// TIA Portal project "KumKoprusu" (V15)

(* hardware
DEVICE "S7-1200 station_1"  S7-1200 Station
   slot 0: "Rack_0"  S7-1200 Rack  Rack  V1.0
   slot 1: "KumKoprusu"  CPU 1214C DC/DC/Rly  6ES7 214-1HG40-0XB0  V4.2
   slot 2: "DI 16x24VDC/DQ 16xRelay_1"  SM 1223 DI16/DQ16 x relay  6ES7 223-1PL32-0XB0  V2.0
*)

// ===== PLC "KumKoprusu"  CPU 1214C DC/DC/Rly =====

VAR_GLOBAL   // PLC tag table "Default tag table"
   "SN_PULS" AT %M2.0 : Bool;
   "SN" AT %MW4 : Int;
   "DK_PULSE" AT %M2.1 : Bool;
END_VAR

VAR_GLOBAL   // PLC tag table "Input"
   "KPR_ACLSTP" AT %I0.0 : Bool;
   "KPR_ILERI_MAN/OTO" AT %I0.1 : Bool;
   "KPR_GERI_MAN/OTO" AT %I0.4 : Bool;
   "KPR_BASTA" AT %I0.7 : Bool;
   "KPR_SONDA" AT %I1.0 : Bool;
   "SYR1_MAN/OTO" AT %I1.1 : Bool;
   "SYR1_YKRD" AT %I1.4 : Bool;
   "SYR1_ASGD" AT %I1.5 : Bool;
   "SYR2_MAN/OTO" AT %I2.0 : Bool;
   "SYR2_YKRD" AT %I2.3 : Bool;
   "SYR2_ASGD" AT %I2.4 : Bool;
   "KPR_GERI_ARZ" AT %I0.6 : Bool;
   "P1_MAN/OTO" AT %I2.5 : Bool;
   "P1_DVRD" AT %I2.6 : Bool;
   "P1_ARZ" AT %I2.7 : Bool;
   "P2_MAN/OTO" AT %I3.0 : Bool;
   "P2_DVRD" AT %I3.1 : Bool;
   "P2_ARZ" AT %I3.2 : Bool;
   "SYR1_DVRD" AT %I1.2 : Bool;
   "SYR1_ARZ" AT %I1.3 : Bool;
   "SYR2_DVRD" AT %I2.1 : Bool;
   "SYR2_ARZ" AT %I2.2 : Bool;
   "KPR_ILERI_ARZ" AT %I0.3 : Bool;
   "KPR_ILERI_DVRD" AT %I0.2 : Bool;
   "KPR_GERI_DVRD" AT %I0.5 : Bool;
END_VAR

VAR_GLOBAL   // PLC tag table "Output"
   "KPR_ILERI_RUNQ" AT %Q0.0 : Bool;
   "KPR_GERI_RUNQ" AT %Q0.1 : Bool;
   "SYR1_ASG_RUNQ" AT %Q0.2 : Bool;
   "SYR1_YKR_RUNQ" AT %Q0.3 : Bool;
   "SYR2_ASG_RUNQ" AT %Q0.4 : Bool;
   "SYR2_YKR_RUNQ" AT %Q0.5 : Bool;
   "P1_RUNQ" AT %Q1.0 : Bool;
   "P2_RUNQ" AT %Q1.1 : Bool;
END_VAR

VAR_GLOBAL   // PLC tag table "Flag"
   "System_Byte" AT %MB1 : Byte;
   "FirstScan" AT %M1.0 : Bool;
   "DiagStatusUpdate" AT %M1.1 : Bool;
   "AlwaysTRUE" AT %M1.2 : Bool;
   "AlwaysFALSE" AT %M1.3 : Bool;
   "Clock_Byte" AT %MB0 : Byte;
   "Clock_10Hz" AT %M0.0 : Bool;
   "Clock_5Hz" AT %M0.1 : Bool;
   "Clock_2.5Hz" AT %M0.2 : Bool;
   "Clock_2Hz" AT %M0.3 : Bool;
   "Clock_1.25Hz" AT %M0.4 : Bool;
   "Clock_1Hz" AT %M0.5 : Bool;
   "Clock_0.625Hz" AT %M0.6 : Bool;
   "Clock_0.5Hz" AT %M0.7 : Bool;
END_VAR

// folder: DB

DATA_BLOCK "KOPRU_DB"   // DB1
{ S7_Optimized_Access := 'TRUE' }
VERSION : 0.1
// stored: InstanceOfName KOPRU_FB
"KOPRU_FB"
BEGIN
END_DATA_BLOCK

DATA_BLOCK "FB_I/O"   // DB2
{ S7_Optimized_Access := 'FALSE' }
VERSION : 0.1
   VAR
      KPR_SCD_RESET : Bool;
      "KPR_SCD_MAN/OTO" : Bool;
      KPR_SCD_MAN_İLERİ : Bool;
      KPR_SCD_MAN_GERİ : Bool;
      SYR_SCD_RESET : Bool;
      "SYR1_SCD_MAN/OTO" : Bool;
      SYR1_SCD_MAN_ASAGI : Bool;
      SYR1_SCD_MAN_YUKARI : Bool;
      "SYR2_SCD_MAN/OTO" : Bool;
      SYR2_SCD_MAN_ASAGI : Bool;
      SYR2_SCD_MAN_YUKARI : Bool;
      "P1_SCD_MAN/OTO" : Bool;
      P1_SCD_MAN_CALIS : Bool;
      "P2_SCD_MAN/OTO" : Bool;
      P2_SCD_MAN_CALIS : Bool;
      Q_KPR_ACIL_STOP : Bool;
      Q_KPR_OTO : Bool;
      Q_KPR_ILERI_GDYR : Bool;
      Q_KPR_SONDA : Bool;
      Q_KPR_GERI_GDYR : Bool;
      Q_KPR_BASTA : Bool;
      Q_KPR_ARIZA : Bool;
      Q_KPR_GECIKME_HATA : Bool;
      Q_KPR_SWITCH_HATA : Bool;
      Q_SYR1_OTO : Bool;
      Q_SYR1_DVRD : Bool;
      Q_SYR1_ASAGIDA : Bool;
      Q_SYR1_YUKARIDA : Bool;
      Q_SYR1_ARIZA : Bool;
      Q_SYR1_GECIKME_HATA : Bool;
      Q_SYR1_SWITCH_HATA : Bool;
      Q_SYR2_OTO : Bool;
      Q_SYR2_DVRD : Bool;
      Q_SYR2_ASAGIDA : Bool;
      Q_SYR2_YUKARIDA : Bool;
      Q_SYR2_ARIZA : Bool;
      Q_SYR2_GECIKME_HATA : Bool;
      Q_SYR2_SWITCH_HATA : Bool;
      Q_P1_OTO : Bool;
      Q_P1_CALISIYOR : Bool;
      Q_P1_ARIZA : Bool;
      Q_P2_OTO : Bool;
      Q_P2_CALISIYOR : Bool;
      Q_P2_ARIZA : Bool;
      Q_PARK_KALAN_SURE : Int;
      Q_IST_KALAN_SURE : Int;
      Q_KPR_SAAT : DInt;
      Q_KPR_DK : DInt;
      Q_KPR_BAKIM_ZAM_FARK : DInt;
      Q_SYR1_SAAT : DInt;
      Q_SYR1_DK : DInt;
      Q_SYR1_BAKIM_ZAM_FARK : DInt;
      Q_SYR2_SAAT : DInt;
      Q_SYR2_DK : DInt;
      Q_SYR2_BAKIM_ZAM_FARK : DInt;
   END_VAR
BEGIN
END_DATA_BLOCK

// folder: (top level)

ORGANIZATION_BLOCK "Main"   // OB1, LAD, ProgramCycle
TITLE = "Main Program Sweep (Cycle)"
{ S7_Optimized_Access := 'TRUE' }
VERSION : 0.1
   VAR_INPUT
      Initial_Call : Bool;   // Initial call of this OB
      Remanence : Bool;   // =True, if remanent data are available
   END_VAR
   VAR_TEMP   // added for the SCL form of the ladder/FBD networks
      _w1 : Bool;
      _w2 : Bool;
   END_VAR
BEGIN

REGION Network 1
   // SN PULSE
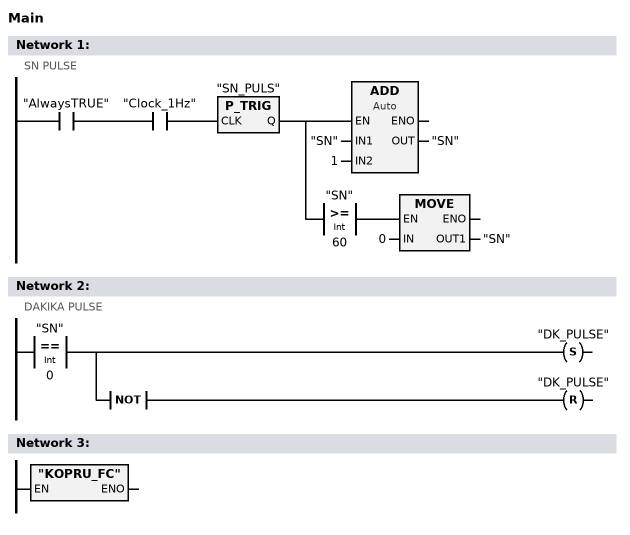
   RUNG wire#powerrail
      Contact( "AlwaysTRUE" )
      Contact( "Clock_1Hz" )
      P_Trig( "SN_PULS" )
      wire#w1
      Add(in1 := "SN", in2 := 1, out => "SN")
   END_RUNG
   RUNG wire#w1
      { S7_Templates := "SrcType := Int" } GE_Contact(in1 := "SN", in2 := 60)
      Move(in := 0, out1 => "SN")
   END_RUNG
   // the same network as SCL:
   #_w1 := "AlwaysTRUE" AND "Clock_1Hz";
   #_w2 := #_w1 AND NOT "SN_PULS";   // rising edge
   "SN_PULS" := #_w1;
   IF #_w2 THEN "SN" := "SN" + 1; END_IF;
   IF #_w2 AND ("SN" >= 60) THEN "SN" := 0; END_IF;
END_REGION

REGION Network 2
   // DAKIKA PULSE
   RUNG wire#powerrail
      { S7_Templates := "SrcType := Int" } EQ_Contact(in1 := "SN", in2 := 0)
      wire#w1
      S_Coil( "DK_PULSE" )
   END_RUNG
   RUNG wire#w1
      Not()
      R_Coil( "DK_PULSE" )
   END_RUNG
   // the same network as SCL:
   #_w1 := "SN" = 0;
   IF #_w1 THEN "DK_PULSE" := TRUE; END_IF;
   IF NOT #_w1 THEN "DK_PULSE" := FALSE; END_IF;
END_REGION

REGION Network 3
   RUNG wire#powerrail
      "KOPRU_FC"()
   END_RUNG
   // the same network as SCL:
   "KOPRU_FC"();
END_REGION
END_ORGANIZATION_BLOCK

// folder: FB

FUNCTION_BLOCK "KOPRU_FB"   // FB1, LAD
{ S7_Optimized_Access := 'TRUE' }
VERSION : 0.1
   VAR_INPUT
      KPR_ACLSTP : Bool;
      KPR_RESET : Bool;
      "KPR_SCADA_MAN/OTO" : Bool;
      "KPR_ILERI_MAN/OTO" : Bool;
      KPR_ILERI_DVRD : Bool;
      KPR_ILERI_ARZ : Bool;
      "KPR_GERI_MAN/OTO" : Bool;
      KPR_GERI_DVRD : Bool;
      KPR_GERI_ARZ : Bool;
      KPR_BASTA : Bool;
      KPR_SONDA : Bool;
      KPR_MAN_İLERİ : Bool;
      KPR_MAN_GERİ : Bool;
      KPR_BAKIM_ZAM_SET : DInt;
      SYR_RESET : Bool;
      "SYR1_SCADA_MAN/OTO" : Bool;
      "SYR1_MAN/OTO" : Bool;
      SYR1_DVRD : Bool;
      SYR1_ARZ : Bool;
      SYR1_YKRD : Bool;
      SYR1_ASGD : Bool;
      SYR1_MAN_ASAGI : Bool;
      SYR1_MAN_YUKARI : Bool;
      "SYR2_SCADA_MAN/OTO" : Bool;
      "SYR2_MAN/OTO" : Bool;
      SYR2_DVRD : Bool;
      SYR2_ARZ : Bool;
      SYR2_YKRD : Bool;
      SYR2_ASGD : Bool;
      SYR2_MAN_ASAGI : Bool;
      SYR2_MAN_YUKARI : Bool;
      SYR_BAKIM_ZAM_SET : DInt;
      "P1_SCADA_MAN/OTO" : Bool;
      "P1_MAN/OTO" : Bool;
      P1_DVRD : Bool;
      P1_ARZ : Bool;
      P1_MAN_CALIS : Bool;
      "P2_SCADA_MAN/OTO" : Bool;
      "P2_MAN/OTO" : Bool;
      P2_DVRD : Bool;
      P2_ARZ : Bool;
      P2_MAN_CALIS : Bool;
      DAKIKA_PULSE : Bool;
      SANIYE_PULSE : Bool;
      "PARK_BEKLEME_SURESI(DK)" : Int;
      "ISTASYON_BEKLEME_SURESI(DK)" : Int;
      "GECIKME_HATASI(SN)" : Int;
   END_VAR
   VAR_OUTPUT
      Q_KPR_ACIL_STOP : Bool;
      Q_KPR_OTO : Bool;
      Q_KPR_ILERI_GIT : Bool;
      Q_KPR_GERI_GIT : Bool;
      Q_KPR_ILERI_GDYR : Bool;
      Q_KPR_SONDA : Bool;
      Q_KPR_GERI_GDYR : Bool;
      Q_KPR_BASTA : Bool;
      Q_KPR_ARIZA : Bool;
      Q_KPR_GECIKME_HATA : Bool;
      Q_KPR_SWITCH_HATA : Bool;
      Q_SYR1_OTO : Bool;
      Q_SYR1_ASAGI_GIT : Bool;
      Q_SYR1_YUKARI_GIT : Bool;
      Q_SYR1_DVRD : Bool;
      Q_SYR1_ASAGIDA : Bool;
      Q_SYR1_YUKARIDA : Bool;
      Q_SYR1_ARIZA : Bool;
      Q_SYR1_GECIKME_HATA : Bool;
      Q_SYR1_SWITCH_HATA : Bool;
      Q_SYR2_OTO : Bool;
      Q_SYR2_ASAGI_GIT : Bool;
      Q_SYR2_YUKARI_GIT : Bool;
      Q_SYR2_DVRD : Bool;
      Q_SYR2_ASAGIDA : Bool;
      Q_SYR2_YUKARIDA : Bool;
      Q_SYR2_ARIZA : Bool;
      Q_SYR2_GECIKME_HATA : Bool;
      Q_SYR2_SWITCH_HATA : Bool;
      Q_P1_OTO : Bool;
      Q_P1_CALIS : Bool;
      Q_P1_CALISIYOR : Bool;
      Q_P1_ARIZA : Bool;
      Q_P2_OTO : Bool;
      Q_P2_CALIS : Bool;
      Q_P2_CALISIYOR : Bool;
      Q_P2_ARIZA : Bool;
      Q_PARK_KALAN_SURE : Int;
      Q_IST_KALAN_SURE : Int;
      Q_KPR_SAAT : DInt;
      Q_KPR_DK : DInt;
      Q_KPR_BAKIM_ZAM_FARK : DInt;
      Q_SYR1_BAKIM_ZAM_FARK : DInt;
      Q_SYR1_SAAT : DInt;
      Q_SYR1_DK : DInt;
      Q_SYR2_BAKIM_ZAM_FARK : DInt;
      Q_SYR2_SAAT : DInt;
      Q_SYR2_DK : DInt;
   END_VAR
   VAR
      ALWAYS_ON : Bool;
      SISTEM_OTO_CLSBLR : Bool;
      SISTEM_OTO : Bool;
      "KPR_MAN/OTO" : Bool;
      KPR_ARIZA : Bool;
      KPR_GENEL_HATA : Bool;
      ILERI_GIT : Bool;
      GERI_GIT : Bool;
      ASAGI_GIT : Bool;
      YUKARI_GIT : Bool;
      "SYR_SCADA_MAN/OTO" : Bool;
      "SYR_MAN/OTO" : Bool;
      PARK_SURE_OK : Bool;
      PARK_SURE : Int;
      SYR1_ZAMAN : Int;
      KPR_ZAMAN : Int;
      SYR_GENEL_HATA : Bool;
      NEGATIF_KENAR_1 : Bool;
      NEGATIF_KENAR_2 : Bool;
      NEGATIF_KENAR_3 : Bool;
      NEGATIF_KENAR_4 : Bool;
      NEGATIF_KENAR_5 : Bool;
      POZ_1 : Bool;
      POZ_2 : Bool;
      POZ_3 : Bool;
      SAAT : DInt;
      DAKIKA : DInt;
      SANIYE : DInt;
      SAAT_1 : DInt;
      DAKIKA_1 : DInt;
      SANIYE_1 : DInt;
      SAAT_2 : DInt;
      DAKIKA_2 : DInt;
      SANIYE_2 : DInt;
      ISTASYON_SURE : Int;
      IST_SURE_OK : Bool;
      P2_CALIS : Bool;
      P1_CALIS : Bool;
   END_VAR
   VAR_TEMP
      KPR_CALISYOR : Bool;
      KPR_ILERI_CALIS : Bool;
      KPR_GERI_CALIS : Bool;
      SYR_CALISIYOR : Bool;
      SYR_ASAGIDA : Bool;
      SYR_YUKARDA : Bool;
      SYR1_ASAGI_CALIS : Bool;
      SYR1_YUKARI_CALIS : Bool;
      SYR2_ASAGI_CALIS : Bool;
      SYR2_YUKARI_CALIS : Bool;
      KPR_SWITCH_HATA : Bool;
      SYR1_SWITCH_HATA : Bool;
      SYR2_SWITCH_HATA : Bool;
      KPR_GECIKME_HATA : Bool;
      SYR1_GECIKME_HATA : Bool;
      SYR2_GECIKME_HATA : Bool;
      IPTAL_BITI : Bool;
      SYR2_ZAMAN : DInt;
   END_VAR
   VAR_TEMP   // added for the SCL form of the ladder/FBD networks
      _w1 : Bool;
      _w2 : Bool;
      _w3 : Bool;
   END_VAR
BEGIN

REGION Network 1
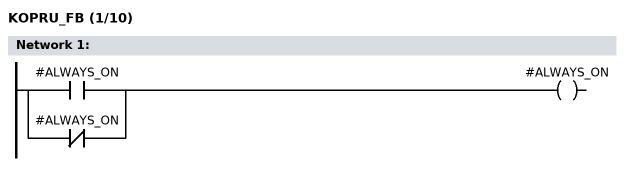
   RUNG wire#powerrail
      Contact( #ALWAYS_ON )
      wire#w1
      Coil( #ALWAYS_ON )
   END_RUNG
   RUNG wire#powerrail
      I_Contact( #ALWAYS_ON )
   END_RUNG wire#w1
   // the same network as SCL:
   #ALWAYS_ON := #ALWAYS_ON OR NOT #ALWAYS_ON;
END_REGION

REGION Network 2
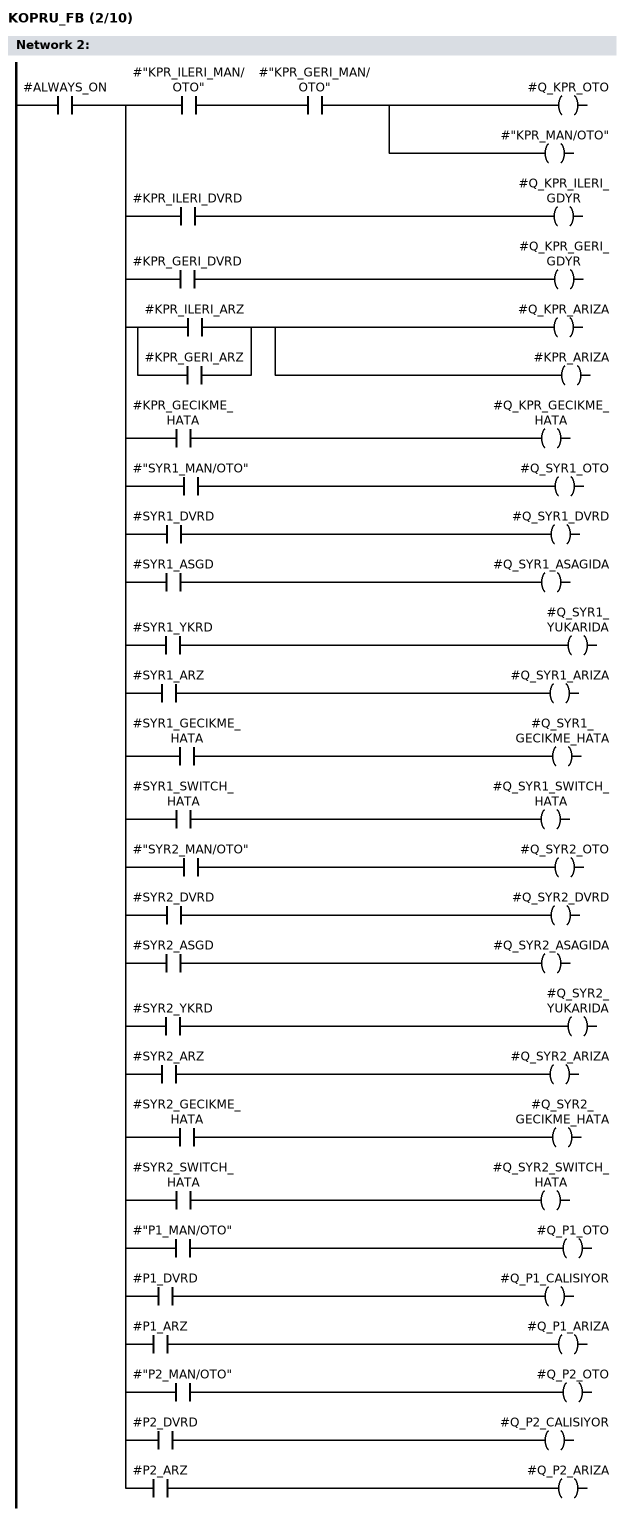
   RUNG wire#powerrail
      Contact( #ALWAYS_ON )
      wire#w1
      Contact( #"KPR_ILERI_MAN/OTO" )
      Contact( #"KPR_GERI_MAN/OTO" )
      wire#w2
      Coil( #Q_KPR_OTO )
   END_RUNG
   RUNG wire#w2
      Coil( #"KPR_MAN/OTO" )
   END_RUNG
   RUNG wire#w1
      Contact( #KPR_ILERI_DVRD )
      Coil( #Q_KPR_ILERI_GDYR )
   END_RUNG
   RUNG wire#w1
      Contact( #KPR_GERI_DVRD )
      Coil( #Q_KPR_GERI_GDYR )
   END_RUNG
   RUNG wire#w1
      Contact( #KPR_ILERI_ARZ )
      wire#w3
      Coil( #Q_KPR_ARIZA )
   END_RUNG
   RUNG wire#w1
      Contact( #KPR_GERI_ARZ )
   END_RUNG wire#w3
   RUNG wire#w3
      Coil( #KPR_ARIZA )
   END_RUNG
   RUNG wire#w1
      Contact( #KPR_GECIKME_HATA )
      Coil( #Q_KPR_GECIKME_HATA )
   END_RUNG
   RUNG wire#w1
      Contact( #"SYR1_MAN/OTO" )
      Coil( #Q_SYR1_OTO )
   END_RUNG
   RUNG wire#w1
      Contact( #SYR1_DVRD )
      Coil( #Q_SYR1_DVRD )
   END_RUNG
   RUNG wire#w1
      Contact( #SYR1_ASGD )
      Coil( #Q_SYR1_ASAGIDA )
   END_RUNG
   RUNG wire#w1
      Contact( #SYR1_YKRD )
      Coil( #Q_SYR1_YUKARIDA )
   END_RUNG
   RUNG wire#w1
      Contact( #SYR1_ARZ )
      Coil( #Q_SYR1_ARIZA )
   END_RUNG
   RUNG wire#w1
      Contact( #SYR1_GECIKME_HATA )
      Coil( #Q_SYR1_GECIKME_HATA )
   END_RUNG
   RUNG wire#w1
      Contact( #SYR1_SWITCH_HATA )
      Coil( #Q_SYR1_SWITCH_HATA )
   END_RUNG
   RUNG wire#w1
      Contact( #"SYR2_MAN/OTO" )
      Coil( #Q_SYR2_OTO )
   END_RUNG
   RUNG wire#w1
      Contact( #SYR2_DVRD )
      Coil( #Q_SYR2_DVRD )
   END_RUNG
   RUNG wire#w1
      Contact( #SYR2_ASGD )
      Coil( #Q_SYR2_ASAGIDA )
   END_RUNG
   RUNG wire#w1
      Contact( #SYR2_YKRD )
      Coil( #Q_SYR2_YUKARIDA )
   END_RUNG
   RUNG wire#w1
      Contact( #SYR2_ARZ )
      Coil( #Q_SYR2_ARIZA )
   END_RUNG
   RUNG wire#w1
      Contact( #SYR2_GECIKME_HATA )
      Coil( #Q_SYR2_GECIKME_HATA )
   END_RUNG
   RUNG wire#w1
      Contact( #SYR2_SWITCH_HATA )
      Coil( #Q_SYR2_SWITCH_HATA )
   END_RUNG
   RUNG wire#w1
      Contact( #"P1_MAN/OTO" )
      Coil( #Q_P1_OTO )
   END_RUNG
   RUNG wire#w1
      Contact( #P1_DVRD )
      Coil( #Q_P1_CALISIYOR )
   END_RUNG
   RUNG wire#w1
      Contact( #P1_ARZ )
      Coil( #Q_P1_ARIZA )
   END_RUNG
   RUNG wire#w1
      Contact( #"P2_MAN/OTO" )
      Coil( #Q_P2_OTO )
   END_RUNG
   RUNG wire#w1
      Contact( #P2_DVRD )
      Coil( #Q_P2_CALISIYOR )
   END_RUNG
   RUNG wire#w1
      Contact( #P2_ARZ )
      Coil( #Q_P2_ARIZA )
   END_RUNG
   // the same network as SCL:
   #Q_KPR_OTO := #ALWAYS_ON AND #"KPR_ILERI_MAN/OTO" AND #"KPR_GERI_MAN/OTO";
   #"KPR_MAN/OTO" := #Q_KPR_OTO;
   #Q_KPR_ILERI_GDYR := #ALWAYS_ON AND #KPR_ILERI_DVRD;
   #Q_KPR_GERI_GDYR := #ALWAYS_ON AND #KPR_GERI_DVRD;
   #Q_KPR_ARIZA := #ALWAYS_ON AND (#KPR_ILERI_ARZ OR #KPR_GERI_ARZ);
   #KPR_ARIZA := #Q_KPR_ARIZA;
   #Q_KPR_GECIKME_HATA := #ALWAYS_ON AND #KPR_GECIKME_HATA;
   #Q_SYR1_OTO := #ALWAYS_ON AND #"SYR1_MAN/OTO";
   #Q_SYR1_DVRD := #ALWAYS_ON AND #SYR1_DVRD;
   #Q_SYR1_ASAGIDA := #ALWAYS_ON AND #SYR1_ASGD;
   #Q_SYR1_YUKARIDA := #ALWAYS_ON AND #SYR1_YKRD;
   #Q_SYR1_ARIZA := #ALWAYS_ON AND #SYR1_ARZ;
   #Q_SYR1_GECIKME_HATA := #ALWAYS_ON AND #SYR1_GECIKME_HATA;
   #Q_SYR1_SWITCH_HATA := #ALWAYS_ON AND #SYR1_SWITCH_HATA;
   #Q_SYR2_OTO := #ALWAYS_ON AND #"SYR2_MAN/OTO";
   #Q_SYR2_DVRD := #ALWAYS_ON AND #SYR2_DVRD;
   #Q_SYR2_ASAGIDA := #ALWAYS_ON AND #SYR2_ASGD;
   #Q_SYR2_YUKARIDA := #ALWAYS_ON AND #SYR2_YKRD;
   #Q_SYR2_ARIZA := #ALWAYS_ON AND #SYR2_ARZ;
   #Q_SYR2_GECIKME_HATA := #ALWAYS_ON AND #SYR2_GECIKME_HATA;
   #Q_SYR2_SWITCH_HATA := #ALWAYS_ON AND #SYR2_SWITCH_HATA;
   #Q_P1_OTO := #ALWAYS_ON AND #"P1_MAN/OTO";
   #Q_P1_CALISIYOR := #ALWAYS_ON AND #P1_DVRD;
   #Q_P1_ARIZA := #ALWAYS_ON AND #P1_ARZ;
   #Q_P2_OTO := #ALWAYS_ON AND #"P2_MAN/OTO";
   #Q_P2_CALISIYOR := #ALWAYS_ON AND #P2_DVRD;
   #Q_P2_ARIZA := #ALWAYS_ON AND #P2_ARZ;
END_REGION

REGION Network 3
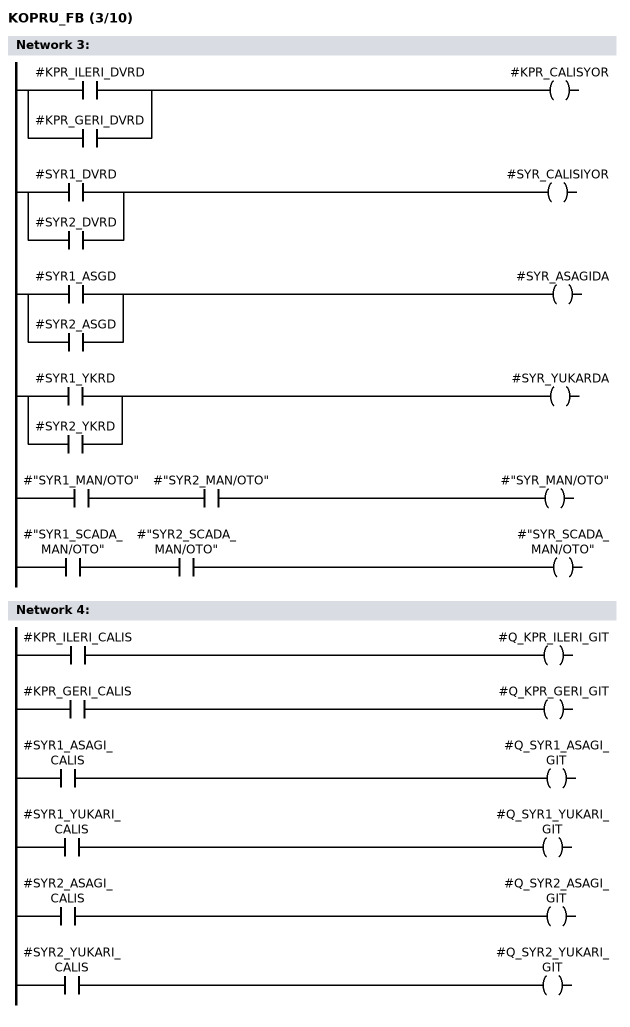
   RUNG wire#powerrail
      Contact( #KPR_ILERI_DVRD )
      wire#w1
      Coil( #KPR_CALISYOR )
   END_RUNG
   RUNG wire#powerrail
      Contact( #KPR_GERI_DVRD )
   END_RUNG wire#w1
   RUNG wire#powerrail
      Contact( #SYR1_DVRD )
      wire#w2
      Coil( #SYR_CALISIYOR )
   END_RUNG
   RUNG wire#powerrail
      Contact( #SYR2_DVRD )
   END_RUNG wire#w2
   RUNG wire#powerrail
      Contact( #SYR1_ASGD )
      wire#w3
      Coil( #SYR_ASAGIDA )
   END_RUNG
   RUNG wire#powerrail
      Contact( #SYR2_ASGD )
   END_RUNG wire#w3
   RUNG wire#powerrail
      Contact( #SYR1_YKRD )
      wire#w4
      Coil( #SYR_YUKARDA )
   END_RUNG
   RUNG wire#powerrail
      Contact( #SYR2_YKRD )
   END_RUNG wire#w4
   RUNG wire#powerrail
      Contact( #"SYR1_MAN/OTO" )
      Contact( #"SYR2_MAN/OTO" )
      Coil( #"SYR_MAN/OTO" )
   END_RUNG
   RUNG wire#powerrail
      Contact( #"SYR1_SCADA_MAN/OTO" )
      Contact( #"SYR2_SCADA_MAN/OTO" )
      Coil( #"SYR_SCADA_MAN/OTO" )
   END_RUNG
   // the same network as SCL:
   #KPR_CALISYOR := #KPR_ILERI_DVRD OR #KPR_GERI_DVRD;
   #SYR_CALISIYOR := #SYR1_DVRD OR #SYR2_DVRD;
   #SYR_ASAGIDA := #SYR1_ASGD OR #SYR2_ASGD;
   #SYR_YUKARDA := #SYR1_YKRD OR #SYR2_YKRD;
   #"SYR_MAN/OTO" := #"SYR1_MAN/OTO" AND #"SYR2_MAN/OTO";
   #"SYR_SCADA_MAN/OTO" := #"SYR1_SCADA_MAN/OTO" AND #"SYR2_SCADA_MAN/OTO";
END_REGION

REGION Network 4
   RUNG wire#powerrail
      Contact( #KPR_ILERI_CALIS )
      Coil( #Q_KPR_ILERI_GIT )
   END_RUNG
   RUNG wire#powerrail
      Contact( #KPR_GERI_CALIS )
      Coil( #Q_KPR_GERI_GIT )
   END_RUNG
   RUNG wire#powerrail
      Contact( #SYR1_ASAGI_CALIS )
      Coil( #Q_SYR1_ASAGI_GIT )
   END_RUNG
   RUNG wire#powerrail
      Contact( #SYR1_YUKARI_CALIS )
      Coil( #Q_SYR1_YUKARI_GIT )
   END_RUNG
   RUNG wire#powerrail
      Contact( #SYR2_ASAGI_CALIS )
      Coil( #Q_SYR2_ASAGI_GIT )
   END_RUNG
   RUNG wire#powerrail
      Contact( #SYR2_YUKARI_CALIS )
      Coil( #Q_SYR2_YUKARI_GIT )
   END_RUNG
   // the same network as SCL:
   #Q_KPR_ILERI_GIT := #KPR_ILERI_CALIS;
   #Q_KPR_GERI_GIT := #KPR_GERI_CALIS;
   #Q_SYR1_ASAGI_GIT := #SYR1_ASAGI_CALIS;
   #Q_SYR1_YUKARI_GIT := #SYR1_YUKARI_CALIS;
   #Q_SYR2_ASAGI_GIT := #SYR2_ASAGI_CALIS;
   #Q_SYR2_YUKARI_GIT := #SYR2_YUKARI_CALIS;
END_REGION

REGION Network 5
   // KÖPRÜ VE SIYIRICI GENEL HATA
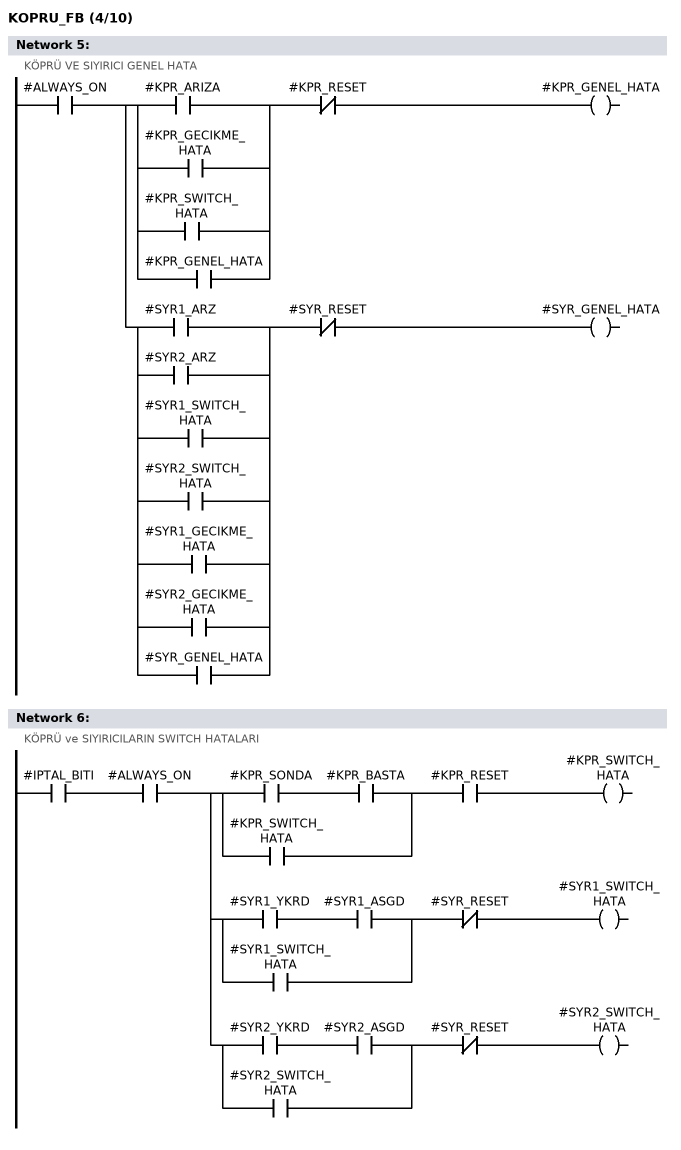
   RUNG wire#powerrail
      Contact( #ALWAYS_ON )
      wire#w1
      Contact( #KPR_ARIZA )
      wire#w2
      I_Contact( #KPR_RESET )
      Coil( #KPR_GENEL_HATA )
   END_RUNG
   RUNG wire#w1
      Contact( #KPR_GECIKME_HATA )
   END_RUNG wire#w2
   RUNG wire#w1
      Contact( #KPR_SWITCH_HATA )
   END_RUNG wire#w2
   RUNG wire#w1
      Contact( #KPR_GENEL_HATA )
   END_RUNG wire#w2
   RUNG wire#w1
      Contact( #SYR1_ARZ )
      wire#w3
      I_Contact( #SYR_RESET )
      Coil( #SYR_GENEL_HATA )
   END_RUNG
   RUNG wire#w1
      Contact( #SYR2_ARZ )
   END_RUNG wire#w3
   RUNG wire#w1
      Contact( #SYR1_SWITCH_HATA )
   END_RUNG wire#w3
   RUNG wire#w1
      Contact( #SYR2_SWITCH_HATA )
   END_RUNG wire#w3
   RUNG wire#w1
      Contact( #SYR1_GECIKME_HATA )
   END_RUNG wire#w3
   RUNG wire#w1
      Contact( #SYR2_GECIKME_HATA )
   END_RUNG wire#w3
   RUNG wire#w1
      Contact( #SYR_GENEL_HATA )
   END_RUNG wire#w3
   // the same network as SCL:
   #KPR_GENEL_HATA := #ALWAYS_ON AND (#KPR_ARIZA OR #KPR_GECIKME_HATA OR #KPR_SWITCH_HATA OR #KPR_GENEL_HATA) AND NOT #KPR_RESET;
   #SYR_GENEL_HATA := #ALWAYS_ON AND (#SYR1_ARZ OR #SYR2_ARZ OR #SYR1_SWITCH_HATA OR #SYR2_SWITCH_HATA OR #SYR1_GECIKME_HATA OR #SYR2_GECIKME_HATA OR #SYR_GENEL_HATA) AND NOT #SYR_RESET;
END_REGION

REGION Network 6
   // KÖPRÜ ve SIYIRICILARIN SWITCH HATALARI
   RUNG wire#powerrail
      Contact( #IPTAL_BITI )
      Contact( #ALWAYS_ON )
      wire#w1
      Contact( #KPR_SONDA )
      Contact( #KPR_BASTA )
      wire#w2
      Contact( #KPR_RESET )
      Coil( #KPR_SWITCH_HATA )
   END_RUNG
   RUNG wire#w1
      Contact( #KPR_SWITCH_HATA )
   END_RUNG wire#w2
   RUNG wire#w1
      Contact( #SYR1_YKRD )
      Contact( #SYR1_ASGD )
      wire#w3
      I_Contact( #SYR_RESET )
      Coil( #SYR1_SWITCH_HATA )
   END_RUNG
   RUNG wire#w1
      Contact( #SYR1_SWITCH_HATA )
   END_RUNG wire#w3
   RUNG wire#w1
      Contact( #SYR2_YKRD )
      Contact( #SYR2_ASGD )
      wire#w4
      I_Contact( #SYR_RESET )
      Coil( #SYR2_SWITCH_HATA )
   END_RUNG
   RUNG wire#w1
      Contact( #SYR2_SWITCH_HATA )
   END_RUNG wire#w4
   // the same network as SCL:
   #_w1 := #IPTAL_BITI AND #ALWAYS_ON;
   #KPR_SWITCH_HATA := #_w1 AND ((#KPR_SONDA AND #KPR_BASTA) OR #KPR_SWITCH_HATA) AND #KPR_RESET;
   #SYR1_SWITCH_HATA := #_w1 AND ((#SYR1_YKRD AND #SYR1_ASGD) OR #SYR1_SWITCH_HATA) AND NOT #SYR_RESET;
   #SYR2_SWITCH_HATA := #_w1 AND ((#SYR2_YKRD AND #SYR2_ASGD) OR #SYR2_SWITCH_HATA) AND NOT #SYR_RESET;
END_REGION

REGION Network 7
   // OTOMATİK ÇALIŞABİLİR İZNİ VE SİSTEM OTO BİLGİSİ
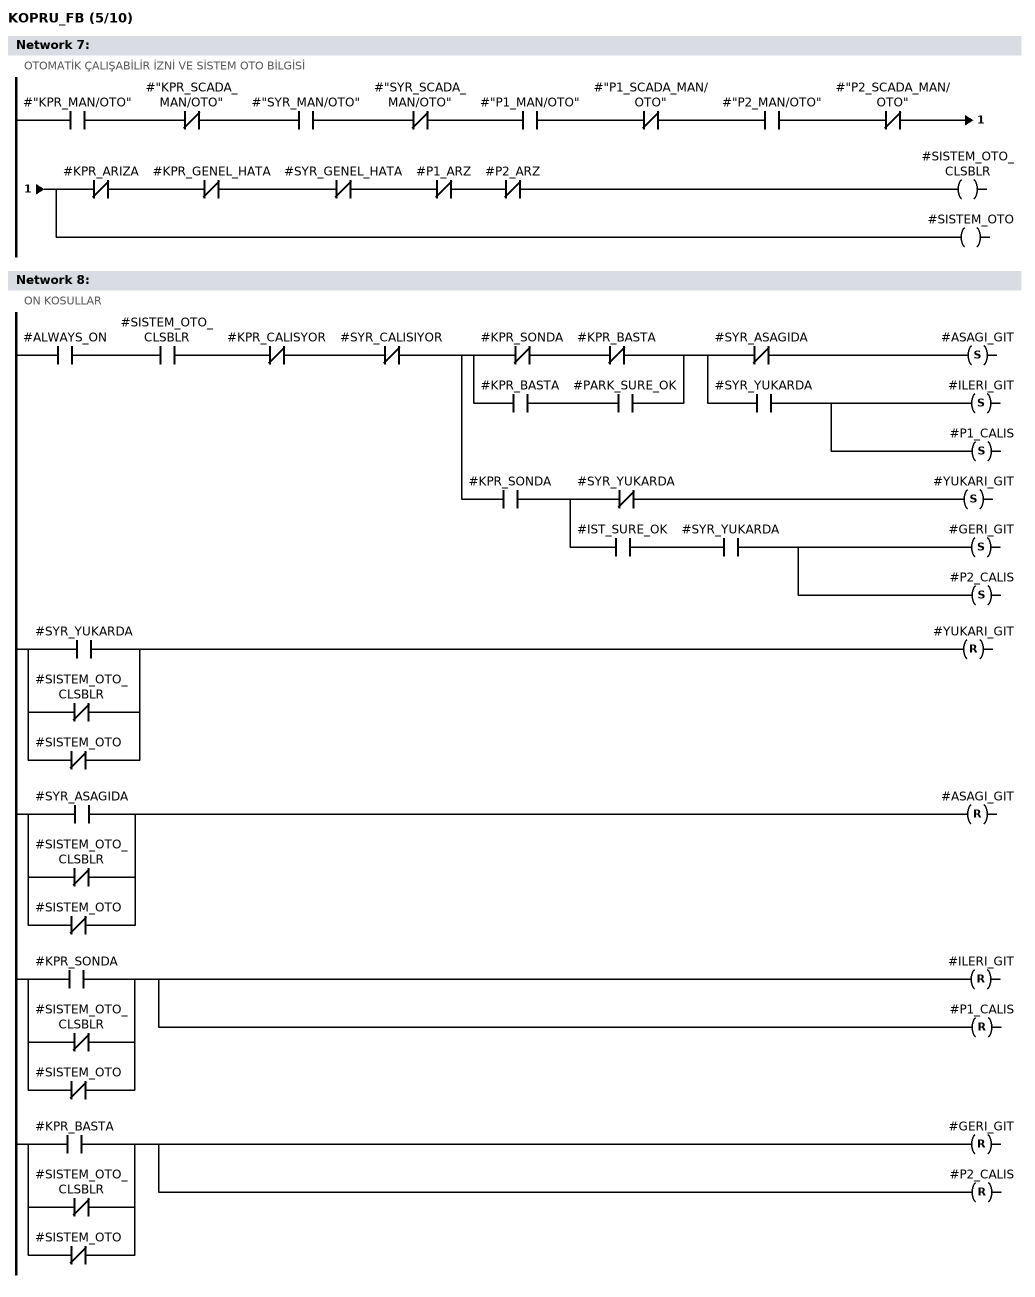
   RUNG wire#powerrail
      Contact( #"KPR_MAN/OTO" )
      I_Contact( #"KPR_SCADA_MAN/OTO" )
      Contact( #"SYR_MAN/OTO" )
      I_Contact( #"SYR_SCADA_MAN/OTO" )
      Contact( #"P1_MAN/OTO" )
      I_Contact( #"P1_SCADA_MAN/OTO" )
      Contact( #"P2_MAN/OTO" )
      I_Contact( #"P2_SCADA_MAN/OTO" )
      wire#w1
      I_Contact( #KPR_ARIZA )
      I_Contact( #KPR_GENEL_HATA )
      I_Contact( #SYR_GENEL_HATA )
      I_Contact( #P1_ARZ )
      I_Contact( #P2_ARZ )
      Coil( #SISTEM_OTO_CLSBLR )
   END_RUNG
   RUNG wire#w1
      Coil( #SISTEM_OTO )
   END_RUNG
   // the same network as SCL:
   #_w1 := #"KPR_MAN/OTO" AND NOT #"KPR_SCADA_MAN/OTO" AND #"SYR_MAN/OTO" AND NOT #"SYR_SCADA_MAN/OTO" AND #"P1_MAN/OTO" AND NOT #"P1_SCADA_MAN/OTO" AND #"P2_MAN/OTO" AND NOT #"P2_SCADA_MAN/OTO";
   #SISTEM_OTO_CLSBLR := #_w1 AND NOT #KPR_ARIZA AND NOT #KPR_GENEL_HATA AND NOT #SYR_GENEL_HATA AND NOT #P1_ARZ AND NOT #P2_ARZ;
   #SISTEM_OTO := #_w1;
END_REGION

REGION Network 8
   // ON KOSULLAR
   RUNG wire#powerrail
      Contact( #ALWAYS_ON )
      Contact( #SISTEM_OTO_CLSBLR )
      I_Contact( #KPR_CALISYOR )
      I_Contact( #SYR_CALISIYOR )
      wire#w1
      I_Contact( #KPR_SONDA )
      I_Contact( #KPR_BASTA )
      wire#w2
      I_Contact( #SYR_ASAGIDA )
      S_Coil( #ASAGI_GIT )
   END_RUNG
   RUNG wire#w1
      Contact( #KPR_BASTA )
      Contact( #PARK_SURE_OK )
   END_RUNG wire#w2
   RUNG wire#w2
      Contact( #SYR_YUKARDA )
      wire#w3
      S_Coil( #ILERI_GIT )
   END_RUNG
   RUNG wire#w3
      S_Coil( #P1_CALIS )
   END_RUNG
   RUNG wire#w1
      Contact( #KPR_SONDA )
      wire#w4
      I_Contact( #SYR_YUKARDA )
      S_Coil( #YUKARI_GIT )
   END_RUNG
   RUNG wire#w4
      Contact( #IST_SURE_OK )
      Contact( #SYR_YUKARDA )
      wire#w5
      S_Coil( #GERI_GIT )
   END_RUNG
   RUNG wire#w5
      S_Coil( #P2_CALIS )
   END_RUNG
   RUNG wire#powerrail
      Contact( #SYR_YUKARDA )
      wire#w6
      R_Coil( #YUKARI_GIT )
   END_RUNG
   RUNG wire#powerrail
      I_Contact( #SISTEM_OTO_CLSBLR )
   END_RUNG wire#w6
   RUNG wire#powerrail
      I_Contact( #SISTEM_OTO )
   END_RUNG wire#w6
   RUNG wire#powerrail
      Contact( #SYR_ASAGIDA )
      wire#w7
      R_Coil( #ASAGI_GIT )
   END_RUNG
   RUNG wire#powerrail
      I_Contact( #SISTEM_OTO_CLSBLR )
   END_RUNG wire#w7
   RUNG wire#powerrail
      I_Contact( #SISTEM_OTO )
   END_RUNG wire#w7
   RUNG wire#powerrail
      Contact( #KPR_SONDA )
      wire#w8
      R_Coil( #ILERI_GIT )
   END_RUNG
   RUNG wire#powerrail
      I_Contact( #SISTEM_OTO_CLSBLR )
   END_RUNG wire#w8
   RUNG wire#powerrail
      I_Contact( #SISTEM_OTO )
   END_RUNG wire#w8
   RUNG wire#w8
      R_Coil( #P1_CALIS )
   END_RUNG
   RUNG wire#powerrail
      Contact( #KPR_BASTA )
      wire#w9
      R_Coil( #GERI_GIT )
   END_RUNG
   RUNG wire#powerrail
      I_Contact( #SISTEM_OTO_CLSBLR )
   END_RUNG wire#w9
   RUNG wire#powerrail
      I_Contact( #SISTEM_OTO )
   END_RUNG wire#w9
   RUNG wire#w9
      R_Coil( #P2_CALIS )
   END_RUNG
   // the same network as SCL:
   #_w1 := #ALWAYS_ON AND #SISTEM_OTO_CLSBLR AND NOT #KPR_CALISYOR AND NOT #SYR_CALISIYOR;
   #_w2 := #_w1 AND ((NOT #KPR_SONDA AND NOT #KPR_BASTA) OR (#KPR_BASTA AND #PARK_SURE_OK));
   IF #_w2 AND NOT #SYR_ASAGIDA THEN #ASAGI_GIT := TRUE; END_IF;
   IF #_w2 AND #SYR_YUKARDA THEN
       #ILERI_GIT := TRUE;
       #P1_CALIS := TRUE;
   END_IF;
   #_w3 := #_w1 AND #KPR_SONDA;
   IF #_w3 AND NOT #SYR_YUKARDA THEN #YUKARI_GIT := TRUE; END_IF;
   IF #_w3 AND #IST_SURE_OK AND #SYR_YUKARDA THEN
       #GERI_GIT := TRUE;
       #P2_CALIS := TRUE;
   END_IF;
   IF #SYR_YUKARDA OR NOT #SISTEM_OTO_CLSBLR OR NOT #SISTEM_OTO THEN #YUKARI_GIT := FALSE; END_IF;
   IF #SYR_ASAGIDA OR NOT #SISTEM_OTO_CLSBLR OR NOT #SISTEM_OTO THEN #ASAGI_GIT := FALSE; END_IF;
   IF #KPR_SONDA OR NOT #SISTEM_OTO_CLSBLR OR NOT #SISTEM_OTO THEN
       #ILERI_GIT := FALSE;
       #P1_CALIS := FALSE;
   END_IF;
   IF #KPR_BASTA OR NOT #SISTEM_OTO_CLSBLR OR NOT #SISTEM_OTO THEN
       #GERI_GIT := FALSE;
       #P2_CALIS := FALSE;
   END_IF;
END_REGION

REGION Network 9
   // KOPRU GERCEK
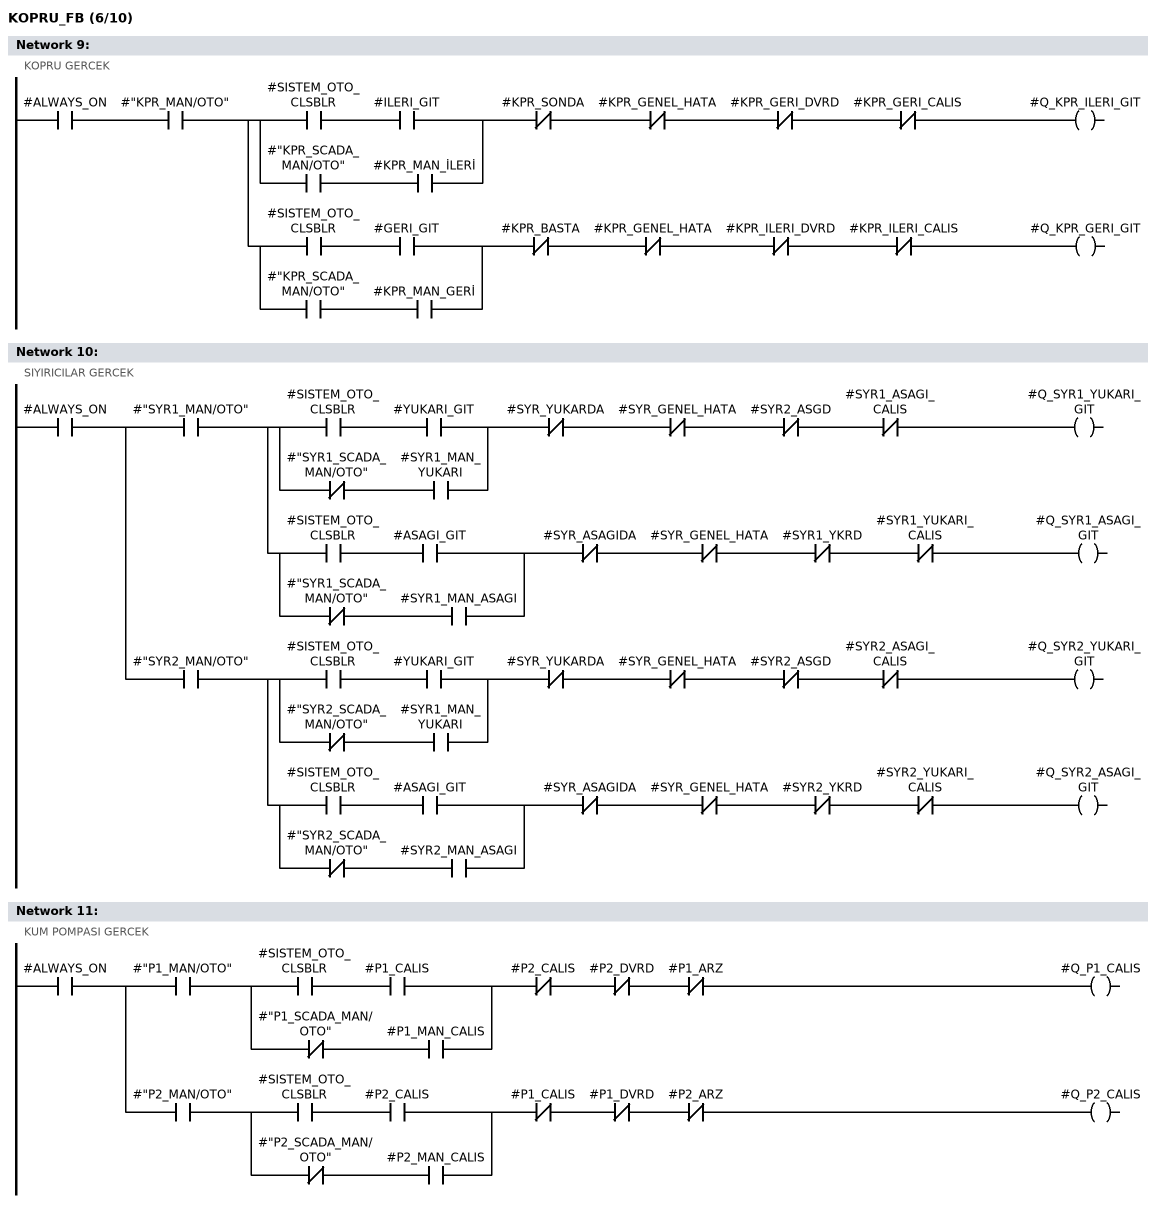
   RUNG wire#powerrail
      Contact( #ALWAYS_ON )
      Contact( #"KPR_MAN/OTO" )
      wire#w1
      Contact( #SISTEM_OTO_CLSBLR )
      Contact( #ILERI_GIT )
      wire#w2
      I_Contact( #KPR_SONDA )
      I_Contact( #KPR_GENEL_HATA )
      I_Contact( #KPR_GERI_DVRD )
      I_Contact( #KPR_GERI_CALIS )
      Coil( #Q_KPR_ILERI_GIT )
   END_RUNG
   RUNG wire#w1
      Contact( #"KPR_SCADA_MAN/OTO" )
      Contact( #KPR_MAN_İLERİ )
   END_RUNG wire#w2
   RUNG wire#w1
      Contact( #SISTEM_OTO_CLSBLR )
      Contact( #GERI_GIT )
      wire#w3
      I_Contact( #KPR_BASTA )
      I_Contact( #KPR_GENEL_HATA )
      I_Contact( #KPR_ILERI_DVRD )
      I_Contact( #KPR_ILERI_CALIS )
      Coil( #Q_KPR_GERI_GIT )
   END_RUNG
   RUNG wire#w1
      Contact( #"KPR_SCADA_MAN/OTO" )
      Contact( #KPR_MAN_GERİ )
   END_RUNG wire#w3
   // the same network as SCL:
   #_w1 := #ALWAYS_ON AND #"KPR_MAN/OTO";
   #Q_KPR_ILERI_GIT := #_w1 AND ((#SISTEM_OTO_CLSBLR AND #ILERI_GIT) OR (#"KPR_SCADA_MAN/OTO" AND #KPR_MAN_İLERİ)) AND NOT #KPR_SONDA AND NOT #KPR_GENEL_HATA AND NOT #KPR_GERI_DVRD AND NOT #KPR_GERI_CALIS;
   #Q_KPR_GERI_GIT := #_w1 AND ((#SISTEM_OTO_CLSBLR AND #GERI_GIT) OR (#"KPR_SCADA_MAN/OTO" AND #KPR_MAN_GERİ)) AND NOT #KPR_BASTA AND NOT #KPR_GENEL_HATA AND NOT #KPR_ILERI_DVRD AND NOT #KPR_ILERI_CALIS;
END_REGION

REGION Network 10
   // SIYIRICILAR GERCEK
   RUNG wire#powerrail
      Contact( #ALWAYS_ON )
      wire#w1
      Contact( #"SYR1_MAN/OTO" )
      wire#w2
      Contact( #SISTEM_OTO_CLSBLR )
      Contact( #YUKARI_GIT )
      wire#w3
      I_Contact( #SYR_YUKARDA )
      I_Contact( #SYR_GENEL_HATA )
      I_Contact( #SYR2_ASGD )
      I_Contact( #SYR1_ASAGI_CALIS )
      Coil( #Q_SYR1_YUKARI_GIT )
   END_RUNG
   RUNG wire#w2
      I_Contact( #"SYR1_SCADA_MAN/OTO" )
      Contact( #SYR1_MAN_YUKARI )
   END_RUNG wire#w3
   RUNG wire#w2
      Contact( #SISTEM_OTO_CLSBLR )
      Contact( #ASAGI_GIT )
      wire#w4
      I_Contact( #SYR_ASAGIDA )
      I_Contact( #SYR_GENEL_HATA )
      I_Contact( #SYR1_YKRD )
      I_Contact( #SYR1_YUKARI_CALIS )
      Coil( #Q_SYR1_ASAGI_GIT )
   END_RUNG
   RUNG wire#w2
      I_Contact( #"SYR1_SCADA_MAN/OTO" )
      Contact( #SYR1_MAN_ASAGI )
   END_RUNG wire#w4
   RUNG wire#w1
      Contact( #"SYR2_MAN/OTO" )
      wire#w5
      Contact( #SISTEM_OTO_CLSBLR )
      Contact( #YUKARI_GIT )
      wire#w6
      I_Contact( #SYR_YUKARDA )
      I_Contact( #SYR_GENEL_HATA )
      I_Contact( #SYR2_ASGD )
      I_Contact( #SYR2_ASAGI_CALIS )
      Coil( #Q_SYR2_YUKARI_GIT )
   END_RUNG
   RUNG wire#w5
      I_Contact( #"SYR2_SCADA_MAN/OTO" )
      Contact( #SYR1_MAN_YUKARI )
   END_RUNG wire#w6
   RUNG wire#w5
      Contact( #SISTEM_OTO_CLSBLR )
      Contact( #ASAGI_GIT )
      wire#w7
      I_Contact( #SYR_ASAGIDA )
      I_Contact( #SYR_GENEL_HATA )
      I_Contact( #SYR2_YKRD )
      I_Contact( #SYR2_YUKARI_CALIS )
      Coil( #Q_SYR2_ASAGI_GIT )
   END_RUNG
   RUNG wire#w5
      I_Contact( #"SYR2_SCADA_MAN/OTO" )
      Contact( #SYR2_MAN_ASAGI )
   END_RUNG wire#w7
   // the same network as SCL:
   #_w1 := #ALWAYS_ON AND #"SYR1_MAN/OTO";
   #Q_SYR1_YUKARI_GIT := #_w1 AND ((#SISTEM_OTO_CLSBLR AND #YUKARI_GIT) OR (NOT #"SYR1_SCADA_MAN/OTO" AND #SYR1_MAN_YUKARI)) AND NOT #SYR_YUKARDA AND NOT #SYR_GENEL_HATA AND NOT #SYR2_ASGD AND NOT #SYR1_ASAGI_CALIS;
   #Q_SYR1_ASAGI_GIT := #_w1 AND ((#SISTEM_OTO_CLSBLR AND #ASAGI_GIT) OR (NOT #"SYR1_SCADA_MAN/OTO" AND #SYR1_MAN_ASAGI)) AND NOT #SYR_ASAGIDA AND NOT #SYR_GENEL_HATA AND NOT #SYR1_YKRD AND NOT #SYR1_YUKARI_CALIS;
   #_w2 := #ALWAYS_ON AND #"SYR2_MAN/OTO";
   #Q_SYR2_YUKARI_GIT := #_w2 AND ((#SISTEM_OTO_CLSBLR AND #YUKARI_GIT) OR (NOT #"SYR2_SCADA_MAN/OTO" AND #SYR1_MAN_YUKARI)) AND NOT #SYR_YUKARDA AND NOT #SYR_GENEL_HATA AND NOT #SYR2_ASGD AND NOT #SYR2_ASAGI_CALIS;
   #Q_SYR2_ASAGI_GIT := #_w2 AND ((#SISTEM_OTO_CLSBLR AND #ASAGI_GIT) OR (NOT #"SYR2_SCADA_MAN/OTO" AND #SYR2_MAN_ASAGI)) AND NOT #SYR_ASAGIDA AND NOT #SYR_GENEL_HATA AND NOT #SYR2_YKRD AND NOT #SYR2_YUKARI_CALIS;
END_REGION

REGION Network 11
   // KUM POMPASI GERCEK
   RUNG wire#powerrail
      Contact( #ALWAYS_ON )
      wire#w1
      Contact( #"P1_MAN/OTO" )
      wire#w2
      Contact( #SISTEM_OTO_CLSBLR )
      Contact( #P1_CALIS )
      wire#w3
      I_Contact( #P2_CALIS )
      I_Contact( #P2_DVRD )
      I_Contact( #P1_ARZ )
      Coil( #Q_P1_CALIS )
   END_RUNG
   RUNG wire#w2
      I_Contact( #"P1_SCADA_MAN/OTO" )
      Contact( #P1_MAN_CALIS )
   END_RUNG wire#w3
   RUNG wire#w1
      Contact( #"P2_MAN/OTO" )
      wire#w4
      Contact( #SISTEM_OTO_CLSBLR )
      Contact( #P2_CALIS )
      wire#w5
      I_Contact( #P1_CALIS )
      I_Contact( #P1_DVRD )
      I_Contact( #P2_ARZ )
      Coil( #Q_P2_CALIS )
   END_RUNG
   RUNG wire#w4
      I_Contact( #"P2_SCADA_MAN/OTO" )
      Contact( #P2_MAN_CALIS )
   END_RUNG wire#w5
   // the same network as SCL:
   #Q_P1_CALIS := #ALWAYS_ON AND #"P1_MAN/OTO" AND ((#SISTEM_OTO_CLSBLR AND #P1_CALIS) OR (NOT #"P1_SCADA_MAN/OTO" AND #P1_MAN_CALIS)) AND NOT #P2_CALIS AND NOT #P2_DVRD AND NOT #P1_ARZ;
   #Q_P2_CALIS := #ALWAYS_ON AND #"P2_MAN/OTO" AND ((#SISTEM_OTO_CLSBLR AND #P2_CALIS) OR (NOT #"P2_SCADA_MAN/OTO" AND #P2_MAN_CALIS)) AND NOT #P1_CALIS AND NOT #P1_DVRD AND NOT #P2_ARZ;
END_REGION

REGION Network 12
   // PARK POZISYONUNDA BEKLEME SURESI
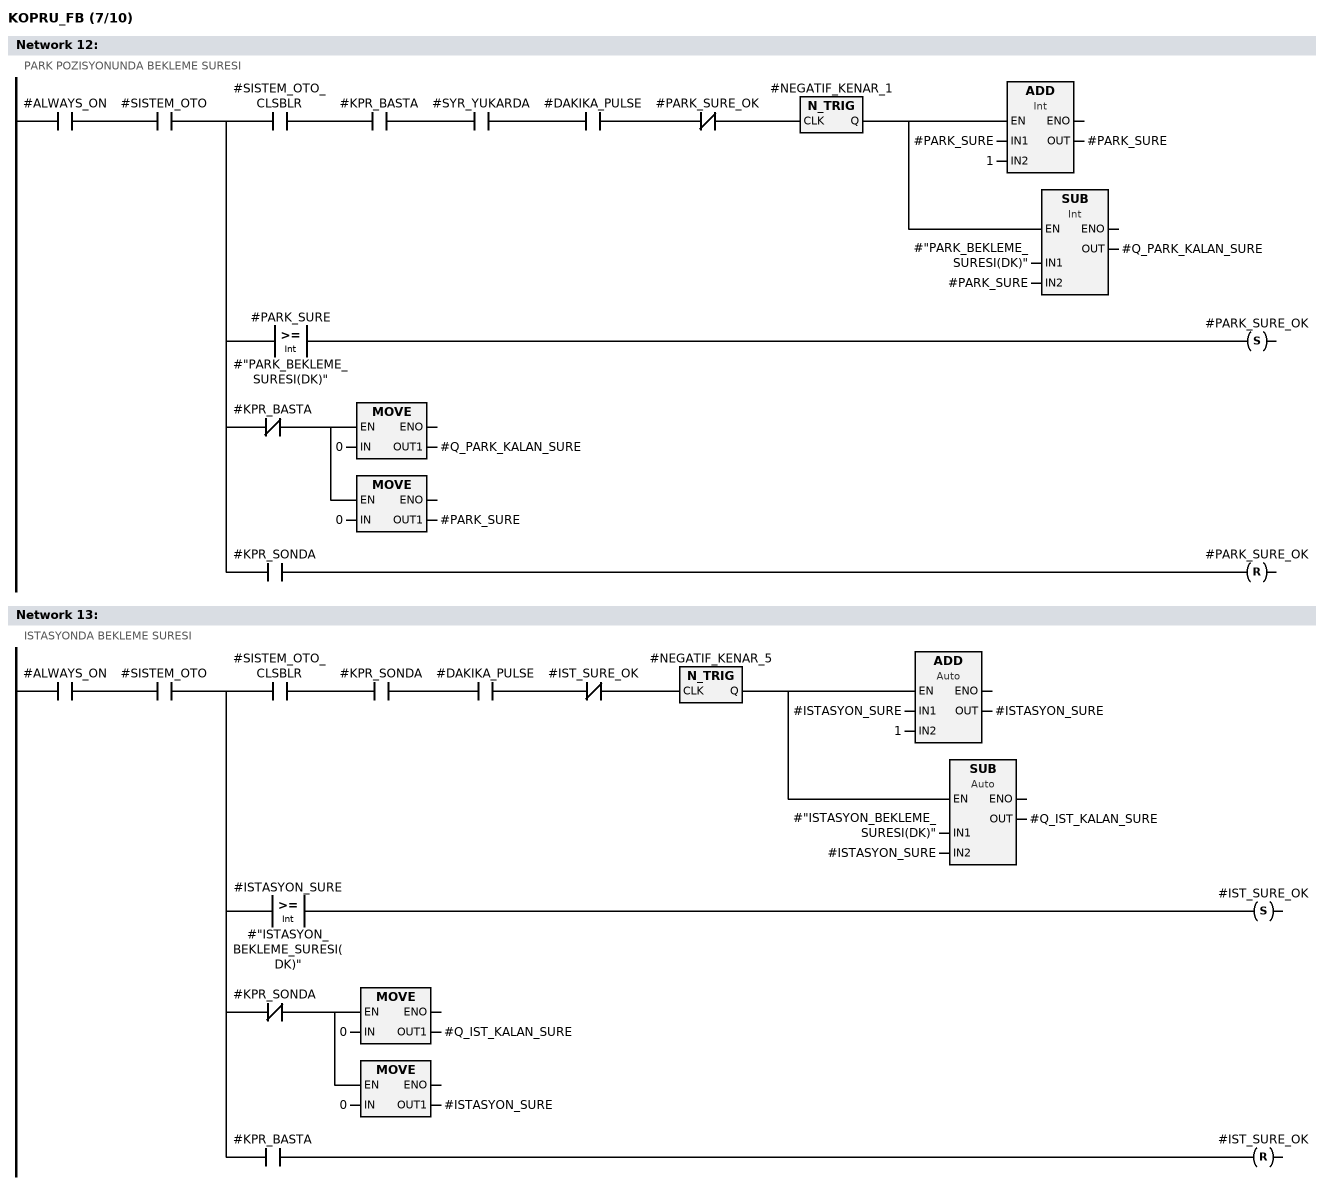
   RUNG wire#powerrail
      Contact( #ALWAYS_ON )
      Contact( #SISTEM_OTO )
      wire#w1
      Contact( #SISTEM_OTO_CLSBLR )
      Contact( #KPR_BASTA )
      Contact( #SYR_YUKARDA )
      Contact( #DAKIKA_PULSE )
      I_Contact( #PARK_SURE_OK )
      N_Trig( #NEGATIF_KENAR_1 )
      wire#w2
      { S7_Templates := "SrcType := Int" } Add(in1 := #PARK_SURE, in2 := 1, out => #PARK_SURE)
   END_RUNG
   RUNG wire#w2
      { S7_Templates := "SrcType := Int" } Sub(in1 := #"PARK_BEKLEME_SURESI(DK)", in2 := #PARK_SURE, out => #Q_PARK_KALAN_SURE)
   END_RUNG
   RUNG wire#w1
      { S7_Templates := "SrcType := Int" } GE_Contact(in1 := #PARK_SURE, in2 := #"PARK_BEKLEME_SURESI(DK)")
      S_Coil( #PARK_SURE_OK )
   END_RUNG
   RUNG wire#w1
      I_Contact( #KPR_BASTA )
      wire#w3
      Move(in := 0, out1 => #Q_PARK_KALAN_SURE)
   END_RUNG
   RUNG wire#w3
      Move(in := 0, out1 => #PARK_SURE)
   END_RUNG
   RUNG wire#w1
      Contact( #KPR_SONDA )
      R_Coil( #PARK_SURE_OK )
   END_RUNG
   // the same network as SCL:
   #_w1 := #ALWAYS_ON AND #SISTEM_OTO;
   #_w2 := #_w1 AND #SISTEM_OTO_CLSBLR AND #KPR_BASTA AND #SYR_YUKARDA AND #DAKIKA_PULSE AND NOT #PARK_SURE_OK;
   #_w3 := NOT #_w2 AND #NEGATIF_KENAR_1;   // falling edge
   #NEGATIF_KENAR_1 := #_w2;
   IF #_w3 THEN
       #PARK_SURE := #PARK_SURE + 1;
       #Q_PARK_KALAN_SURE := #"PARK_BEKLEME_SURESI(DK)" - #PARK_SURE;
   END_IF;
   IF #_w1 AND (#PARK_SURE >= #"PARK_BEKLEME_SURESI(DK)") THEN #PARK_SURE_OK := TRUE; END_IF;
   IF #_w1 AND NOT #KPR_BASTA THEN
       #Q_PARK_KALAN_SURE := 0;
       #PARK_SURE := 0;
   END_IF;
   IF #_w1 AND #KPR_SONDA THEN #PARK_SURE_OK := FALSE; END_IF;
END_REGION

REGION Network 13
   // ISTASYONDA BEKLEME SURESI
   RUNG wire#powerrail
      Contact( #ALWAYS_ON )
      Contact( #SISTEM_OTO )
      wire#w1
      Contact( #SISTEM_OTO_CLSBLR )
      Contact( #KPR_SONDA )
      Contact( #DAKIKA_PULSE )
      I_Contact( #IST_SURE_OK )
      N_Trig( #NEGATIF_KENAR_5 )
      wire#w2
      Add(in1 := #ISTASYON_SURE, in2 := 1, out => #ISTASYON_SURE)
   END_RUNG
   RUNG wire#w2
      Sub(in1 := #"ISTASYON_BEKLEME_SURESI(DK)", in2 := #ISTASYON_SURE, out => #Q_IST_KALAN_SURE)
   END_RUNG
   RUNG wire#w1
      { S7_Templates := "SrcType := Int" } GE_Contact(in1 := #ISTASYON_SURE, in2 := #"ISTASYON_BEKLEME_SURESI(DK)")
      S_Coil( #IST_SURE_OK )
   END_RUNG
   RUNG wire#w1
      I_Contact( #KPR_SONDA )
      wire#w3
      Move(in := 0, out1 => #Q_IST_KALAN_SURE)
   END_RUNG
   RUNG wire#w3
      Move(in := 0, out1 => #ISTASYON_SURE)
   END_RUNG
   RUNG wire#w1
      Contact( #KPR_BASTA )
      R_Coil( #IST_SURE_OK )
   END_RUNG
   // the same network as SCL:
   #_w1 := #ALWAYS_ON AND #SISTEM_OTO;
   #_w2 := #_w1 AND #SISTEM_OTO_CLSBLR AND #KPR_SONDA AND #DAKIKA_PULSE AND NOT #IST_SURE_OK;
   #_w3 := NOT #_w2 AND #NEGATIF_KENAR_5;   // falling edge
   #NEGATIF_KENAR_5 := #_w2;
   IF #_w3 THEN
       #ISTASYON_SURE := #ISTASYON_SURE + 1;
       #Q_IST_KALAN_SURE := #"ISTASYON_BEKLEME_SURESI(DK)" - #ISTASYON_SURE;
   END_IF;
   IF #_w1 AND (#ISTASYON_SURE >= #"ISTASYON_BEKLEME_SURESI(DK)") THEN #IST_SURE_OK := TRUE; END_IF;
   IF #_w1 AND NOT #KPR_SONDA THEN
       #Q_IST_KALAN_SURE := 0;
       #ISTASYON_SURE := 0;
   END_IF;
   IF #_w1 AND #KPR_BASTA THEN #IST_SURE_OK := FALSE; END_IF;
END_REGION

REGION Network 14
   // KOPRU HATA
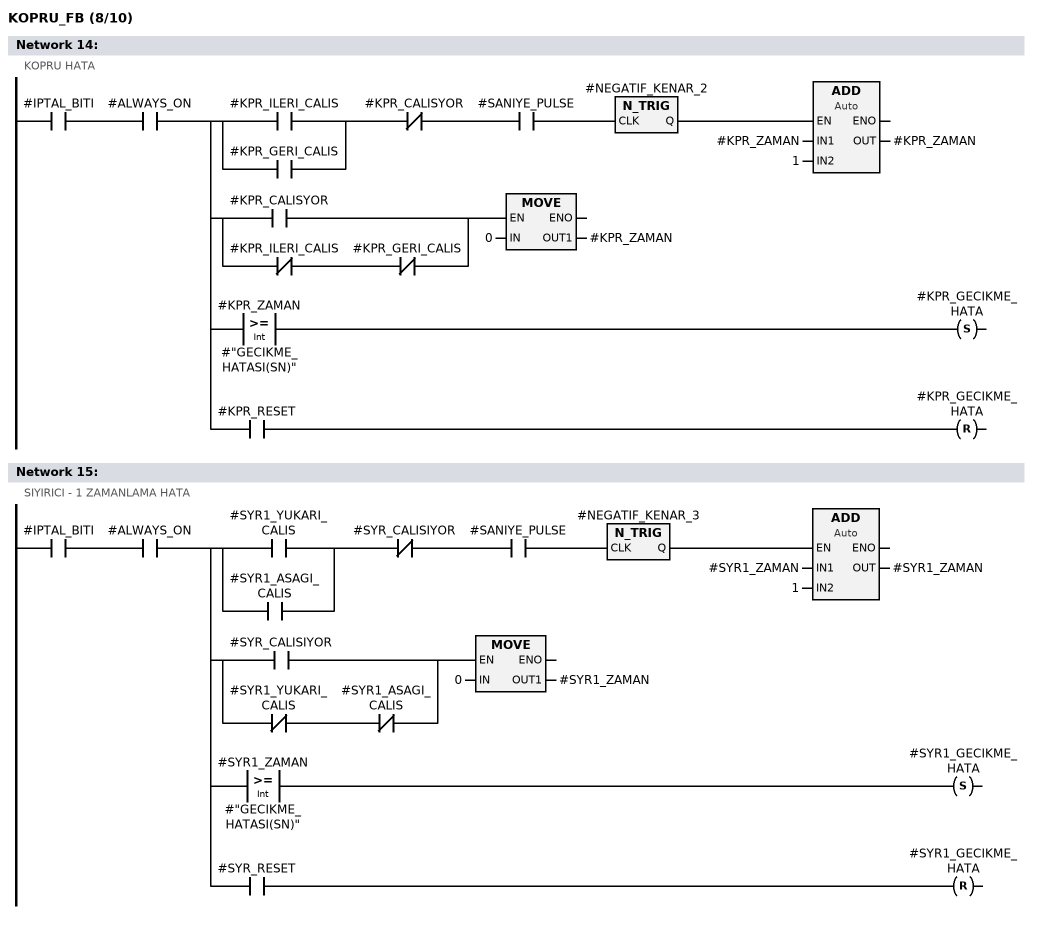
   RUNG wire#powerrail
      Contact( #IPTAL_BITI )
      Contact( #ALWAYS_ON )
      wire#w1
      Contact( #KPR_ILERI_CALIS )
      wire#w2
      I_Contact( #KPR_CALISYOR )
      Contact( #SANIYE_PULSE )
      N_Trig( #NEGATIF_KENAR_2 )
      Add(in1 := #KPR_ZAMAN, in2 := 1, out => #KPR_ZAMAN)
   END_RUNG
   RUNG wire#w1
      Contact( #KPR_GERI_CALIS )
   END_RUNG wire#w2
   RUNG wire#w1
      Contact( #KPR_CALISYOR )
      wire#w3
      Move(in := 0, out1 => #KPR_ZAMAN)
   END_RUNG
   RUNG wire#w1
      I_Contact( #KPR_ILERI_CALIS )
      I_Contact( #KPR_GERI_CALIS )
   END_RUNG wire#w3
   RUNG wire#w1
      { S7_Templates := "SrcType := Int" } GE_Contact(in1 := #KPR_ZAMAN, in2 := #"GECIKME_HATASI(SN)")
      S_Coil( #KPR_GECIKME_HATA )
   END_RUNG
   RUNG wire#w1
      Contact( #KPR_RESET )
      R_Coil( #KPR_GECIKME_HATA )
   END_RUNG
   // the same network as SCL:
   #_w1 := #IPTAL_BITI AND #ALWAYS_ON;
   #_w2 := #_w1 AND (#KPR_ILERI_CALIS OR #KPR_GERI_CALIS) AND NOT #KPR_CALISYOR AND #SANIYE_PULSE;
   #_w3 := NOT #_w2 AND #NEGATIF_KENAR_2;   // falling edge
   #NEGATIF_KENAR_2 := #_w2;
   IF #_w3 THEN #KPR_ZAMAN := #KPR_ZAMAN + 1; END_IF;
   IF #_w1 AND (#KPR_CALISYOR OR (NOT #KPR_ILERI_CALIS AND NOT #KPR_GERI_CALIS)) THEN
       #KPR_ZAMAN := 0;
   END_IF;
   IF #_w1 AND (#KPR_ZAMAN >= #"GECIKME_HATASI(SN)") THEN #KPR_GECIKME_HATA := TRUE; END_IF;
   IF #_w1 AND #KPR_RESET THEN #KPR_GECIKME_HATA := FALSE; END_IF;
END_REGION

REGION Network 15
   // SIYIRICI - 1 ZAMANLAMA HATA
   RUNG wire#powerrail
      Contact( #IPTAL_BITI )
      Contact( #ALWAYS_ON )
      wire#w1
      Contact( #SYR1_YUKARI_CALIS )
      wire#w2
      I_Contact( #SYR_CALISIYOR )
      Contact( #SANIYE_PULSE )
      N_Trig( #NEGATIF_KENAR_3 )
      Add(in1 := #SYR1_ZAMAN, in2 := 1, out => #SYR1_ZAMAN)
   END_RUNG
   RUNG wire#w1
      Contact( #SYR1_ASAGI_CALIS )
   END_RUNG wire#w2
   RUNG wire#w1
      Contact( #SYR_CALISIYOR )
      wire#w3
      Move(in := 0, out1 => #SYR1_ZAMAN)
   END_RUNG
   RUNG wire#w1
      I_Contact( #SYR1_YUKARI_CALIS )
      I_Contact( #SYR1_ASAGI_CALIS )
   END_RUNG wire#w3
   RUNG wire#w1
      { S7_Templates := "SrcType := Int" } GE_Contact(in1 := #SYR1_ZAMAN, in2 := #"GECIKME_HATASI(SN)")
      S_Coil( #SYR1_GECIKME_HATA )
   END_RUNG
   RUNG wire#w1
      Contact( #SYR_RESET )
      R_Coil( #SYR1_GECIKME_HATA )
   END_RUNG
   // the same network as SCL:
   #_w1 := #IPTAL_BITI AND #ALWAYS_ON;
   #_w2 := #_w1 AND (#SYR1_YUKARI_CALIS OR #SYR1_ASAGI_CALIS) AND NOT #SYR_CALISIYOR AND #SANIYE_PULSE;
   #_w3 := NOT #_w2 AND #NEGATIF_KENAR_3;   // falling edge
   #NEGATIF_KENAR_3 := #_w2;
   IF #_w3 THEN #SYR1_ZAMAN := #SYR1_ZAMAN + 1; END_IF;
   IF #_w1 AND (#SYR_CALISIYOR OR (NOT #SYR1_YUKARI_CALIS AND NOT #SYR1_ASAGI_CALIS)) THEN
       #SYR1_ZAMAN := 0;
   END_IF;
   IF #_w1 AND (#SYR1_ZAMAN >= #"GECIKME_HATASI(SN)") THEN #SYR1_GECIKME_HATA := TRUE; END_IF;
   IF #_w1 AND #SYR_RESET THEN #SYR1_GECIKME_HATA := FALSE; END_IF;
END_REGION

REGION Network 16
   // SIYIRICI - 2 ZAMANLAMA HATA
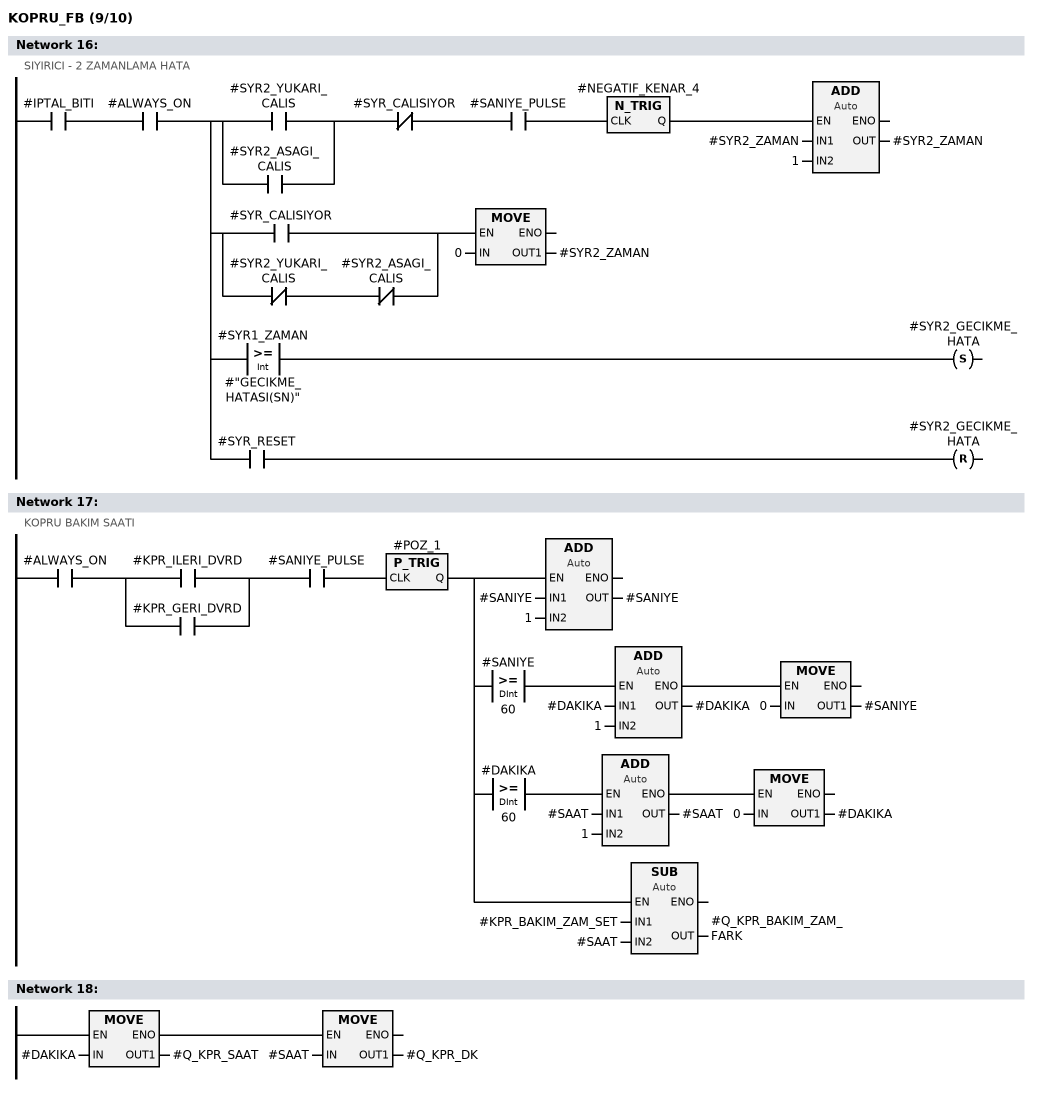
   RUNG wire#powerrail
      Contact( #IPTAL_BITI )
      Contact( #ALWAYS_ON )
      wire#w1
      Contact( #SYR2_YUKARI_CALIS )
      wire#w2
      I_Contact( #SYR_CALISIYOR )
      Contact( #SANIYE_PULSE )
      N_Trig( #NEGATIF_KENAR_4 )
      Add(in1 := #SYR2_ZAMAN, in2 := 1, out => #SYR2_ZAMAN)
   END_RUNG
   RUNG wire#w1
      Contact( #SYR2_ASAGI_CALIS )
   END_RUNG wire#w2
   RUNG wire#w1
      Contact( #SYR_CALISIYOR )
      wire#w3
      Move(in := 0, out1 => #SYR2_ZAMAN)
   END_RUNG
   RUNG wire#w1
      I_Contact( #SYR2_YUKARI_CALIS )
      I_Contact( #SYR2_ASAGI_CALIS )
   END_RUNG wire#w3
   RUNG wire#w1
      { S7_Templates := "SrcType := Int" } GE_Contact(in1 := #SYR1_ZAMAN, in2 := #"GECIKME_HATASI(SN)")
      S_Coil( #SYR2_GECIKME_HATA )
   END_RUNG
   RUNG wire#w1
      Contact( #SYR_RESET )
      R_Coil( #SYR2_GECIKME_HATA )
   END_RUNG
   // the same network as SCL:
   #_w1 := #IPTAL_BITI AND #ALWAYS_ON;
   #_w2 := #_w1 AND (#SYR2_YUKARI_CALIS OR #SYR2_ASAGI_CALIS) AND NOT #SYR_CALISIYOR AND #SANIYE_PULSE;
   #_w3 := NOT #_w2 AND #NEGATIF_KENAR_4;   // falling edge
   #NEGATIF_KENAR_4 := #_w2;
   IF #_w3 THEN #SYR2_ZAMAN := #SYR2_ZAMAN + 1; END_IF;
   IF #_w1 AND (#SYR_CALISIYOR OR (NOT #SYR2_YUKARI_CALIS AND NOT #SYR2_ASAGI_CALIS)) THEN
       #SYR2_ZAMAN := 0;
   END_IF;
   IF #_w1 AND (#SYR1_ZAMAN >= #"GECIKME_HATASI(SN)") THEN #SYR2_GECIKME_HATA := TRUE; END_IF;
   IF #_w1 AND #SYR_RESET THEN #SYR2_GECIKME_HATA := FALSE; END_IF;
END_REGION

REGION Network 17
   // KOPRU BAKIM SAATI
   RUNG wire#powerrail
      Contact( #ALWAYS_ON )
      wire#w1
      Contact( #KPR_ILERI_DVRD )
      wire#w2
      Contact( #SANIYE_PULSE )
      P_Trig( #POZ_1 )
      wire#w3
      Add(in1 := #SANIYE, in2 := 1, out => #SANIYE)
   END_RUNG
   RUNG wire#w1
      Contact( #KPR_GERI_DVRD )
   END_RUNG wire#w2
   RUNG wire#w3
      { S7_Templates := "SrcType := DInt" } GE_Contact(in1 := #SANIYE, in2 := 60)
      Add(in1 := #DAKIKA, in2 := 1, out => #DAKIKA)
      Move(in := 0, out1 => #SANIYE)
   END_RUNG
   RUNG wire#w3
      { S7_Templates := "SrcType := DInt" } GE_Contact(in1 := #DAKIKA, in2 := 60)
      Add(in1 := #SAAT, in2 := 1, out => #SAAT)
      Move(in := 0, out1 => #DAKIKA)
   END_RUNG
   RUNG wire#w3
      Sub(in1 := #KPR_BAKIM_ZAM_SET, in2 := #SAAT, out => #Q_KPR_BAKIM_ZAM_FARK)
   END_RUNG
   // the same network as SCL:
   #_w1 := #ALWAYS_ON AND (#KPR_ILERI_DVRD OR #KPR_GERI_DVRD) AND #SANIYE_PULSE;
   #_w2 := #_w1 AND NOT #POZ_1;   // rising edge
   #POZ_1 := #_w1;
   IF #_w2 THEN #SANIYE := #SANIYE + 1; END_IF;
   IF #_w2 AND (#SANIYE >= 60) THEN
       #DAKIKA := #DAKIKA + 1;
       #SANIYE := 0;
   END_IF;
   IF #_w2 AND (#DAKIKA >= 60) THEN
       #SAAT := #SAAT + 1;
       #DAKIKA := 0;
   END_IF;
   IF #_w2 THEN #Q_KPR_BAKIM_ZAM_FARK := #KPR_BAKIM_ZAM_SET - #SAAT; END_IF;
END_REGION

REGION Network 18
   RUNG wire#powerrail
      Move(in := #DAKIKA, out1 => #Q_KPR_SAAT)
      Move(in := #SAAT, out1 => #Q_KPR_DK)
   END_RUNG
   // the same network as SCL:
   #Q_KPR_SAAT := #DAKIKA;
   #Q_KPR_DK := #SAAT;
END_REGION

REGION Network 19
   // SIYIRICI - 1 BAKIM SAATI
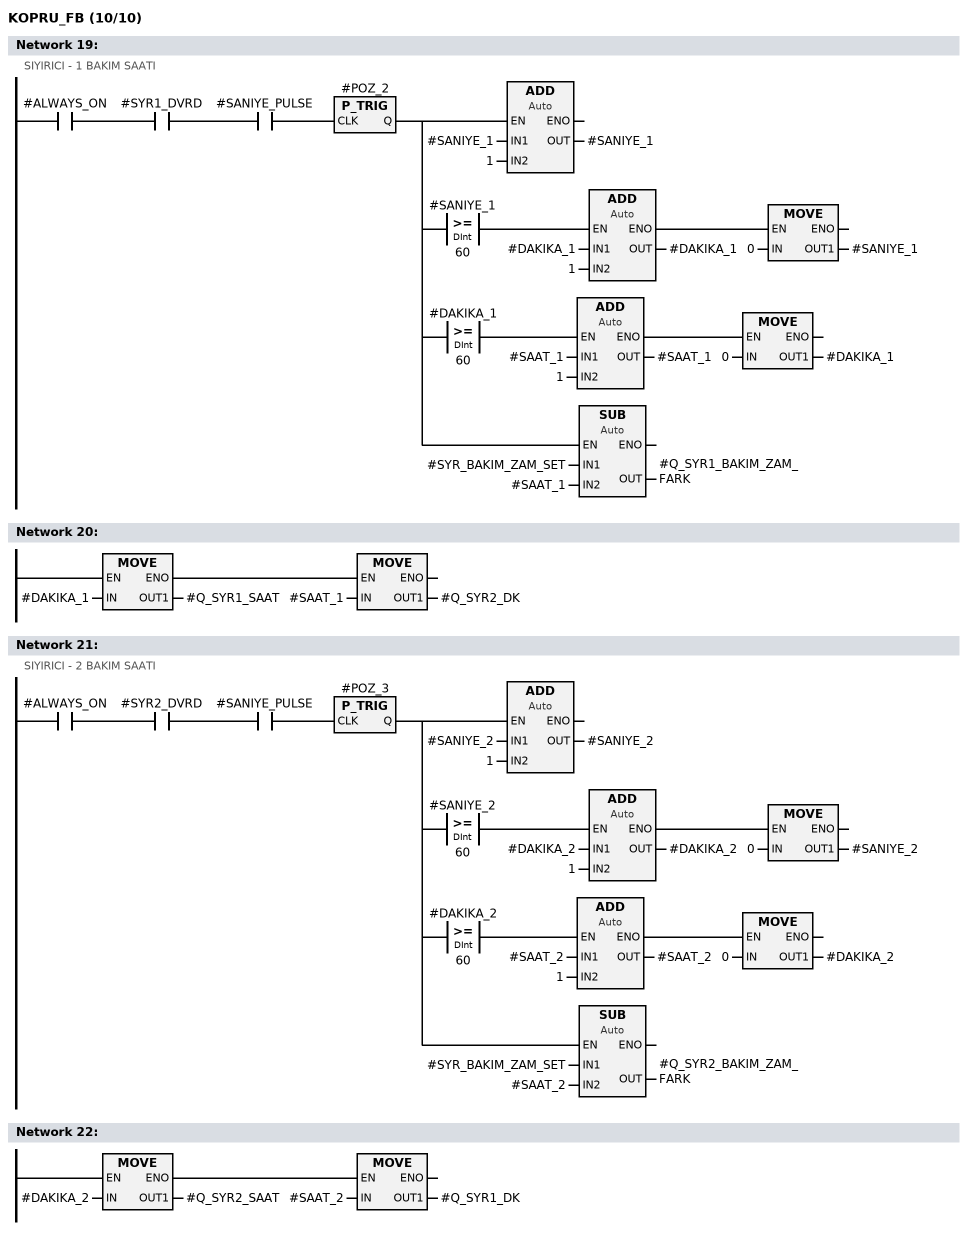
   RUNG wire#powerrail
      Contact( #ALWAYS_ON )
      Contact( #SYR1_DVRD )
      Contact( #SANIYE_PULSE )
      P_Trig( #POZ_2 )
      wire#w1
      Add(in1 := #SANIYE_1, in2 := 1, out => #SANIYE_1)
   END_RUNG
   RUNG wire#w1
      { S7_Templates := "SrcType := DInt" } GE_Contact(in1 := #SANIYE_1, in2 := 60)
      Add(in1 := #DAKIKA_1, in2 := 1, out => #DAKIKA_1)
      Move(in := 0, out1 => #SANIYE_1)
   END_RUNG
   RUNG wire#w1
      { S7_Templates := "SrcType := DInt" } GE_Contact(in1 := #DAKIKA_1, in2 := 60)
      Add(in1 := #SAAT_1, in2 := 1, out => #SAAT_1)
      Move(in := 0, out1 => #DAKIKA_1)
   END_RUNG
   RUNG wire#w1
      Sub(in1 := #SYR_BAKIM_ZAM_SET, in2 := #SAAT_1, out => #Q_SYR1_BAKIM_ZAM_FARK)
   END_RUNG
   // the same network as SCL:
   #_w1 := #ALWAYS_ON AND #SYR1_DVRD AND #SANIYE_PULSE;
   #_w2 := #_w1 AND NOT #POZ_2;   // rising edge
   #POZ_2 := #_w1;
   IF #_w2 THEN #SANIYE_1 := #SANIYE_1 + 1; END_IF;
   IF #_w2 AND (#SANIYE_1 >= 60) THEN
       #DAKIKA_1 := #DAKIKA_1 + 1;
       #SANIYE_1 := 0;
   END_IF;
   IF #_w2 AND (#DAKIKA_1 >= 60) THEN
       #SAAT_1 := #SAAT_1 + 1;
       #DAKIKA_1 := 0;
   END_IF;
   IF #_w2 THEN #Q_SYR1_BAKIM_ZAM_FARK := #SYR_BAKIM_ZAM_SET - #SAAT_1; END_IF;
END_REGION

REGION Network 20
   RUNG wire#powerrail
      Move(in := #DAKIKA_1, out1 => #Q_SYR1_SAAT)
      Move(in := #SAAT_1, out1 => #Q_SYR2_DK)
   END_RUNG
   // the same network as SCL:
   #Q_SYR1_SAAT := #DAKIKA_1;
   #Q_SYR2_DK := #SAAT_1;
END_REGION

REGION Network 21
   // SIYIRICI - 2 BAKIM SAATI
   RUNG wire#powerrail
      Contact( #ALWAYS_ON )
      Contact( #SYR2_DVRD )
      Contact( #SANIYE_PULSE )
      P_Trig( #POZ_3 )
      wire#w1
      Add(in1 := #SANIYE_2, in2 := 1, out => #SANIYE_2)
   END_RUNG
   RUNG wire#w1
      { S7_Templates := "SrcType := DInt" } GE_Contact(in1 := #SANIYE_2, in2 := 60)
      Add(in1 := #DAKIKA_2, in2 := 1, out => #DAKIKA_2)
      Move(in := 0, out1 => #SANIYE_2)
   END_RUNG
   RUNG wire#w1
      { S7_Templates := "SrcType := DInt" } GE_Contact(in1 := #DAKIKA_2, in2 := 60)
      Add(in1 := #SAAT_2, in2 := 1, out => #SAAT_2)
      Move(in := 0, out1 => #DAKIKA_2)
   END_RUNG
   RUNG wire#w1
      Sub(in1 := #SYR_BAKIM_ZAM_SET, in2 := #SAAT_2, out => #Q_SYR2_BAKIM_ZAM_FARK)
   END_RUNG
   // the same network as SCL:
   #_w1 := #ALWAYS_ON AND #SYR2_DVRD AND #SANIYE_PULSE;
   #_w2 := #_w1 AND NOT #POZ_3;   // rising edge
   #POZ_3 := #_w1;
   IF #_w2 THEN #SANIYE_2 := #SANIYE_2 + 1; END_IF;
   IF #_w2 AND (#SANIYE_2 >= 60) THEN
       #DAKIKA_2 := #DAKIKA_2 + 1;
       #SANIYE_2 := 0;
   END_IF;
   IF #_w2 AND (#DAKIKA_2 >= 60) THEN
       #SAAT_2 := #SAAT_2 + 1;
       #DAKIKA_2 := 0;
   END_IF;
   IF #_w2 THEN #Q_SYR2_BAKIM_ZAM_FARK := #SYR_BAKIM_ZAM_SET - #SAAT_2; END_IF;
END_REGION

REGION Network 22
   RUNG wire#powerrail
      Move(in := #DAKIKA_2, out1 => #Q_SYR2_SAAT)
      Move(in := #SAAT_2, out1 => #Q_SYR1_DK)
   END_RUNG
   // the same network as SCL:
   #Q_SYR2_SAAT := #DAKIKA_2;
   #Q_SYR1_DK := #SAAT_2;
END_REGION
END_FUNCTION_BLOCK

// folder: FC

FUNCTION "KOPRU_FC" : Void   // FC1, LAD
{ S7_Optimized_Access := 'TRUE' }
VERSION : 0.1
BEGIN

REGION Network 1
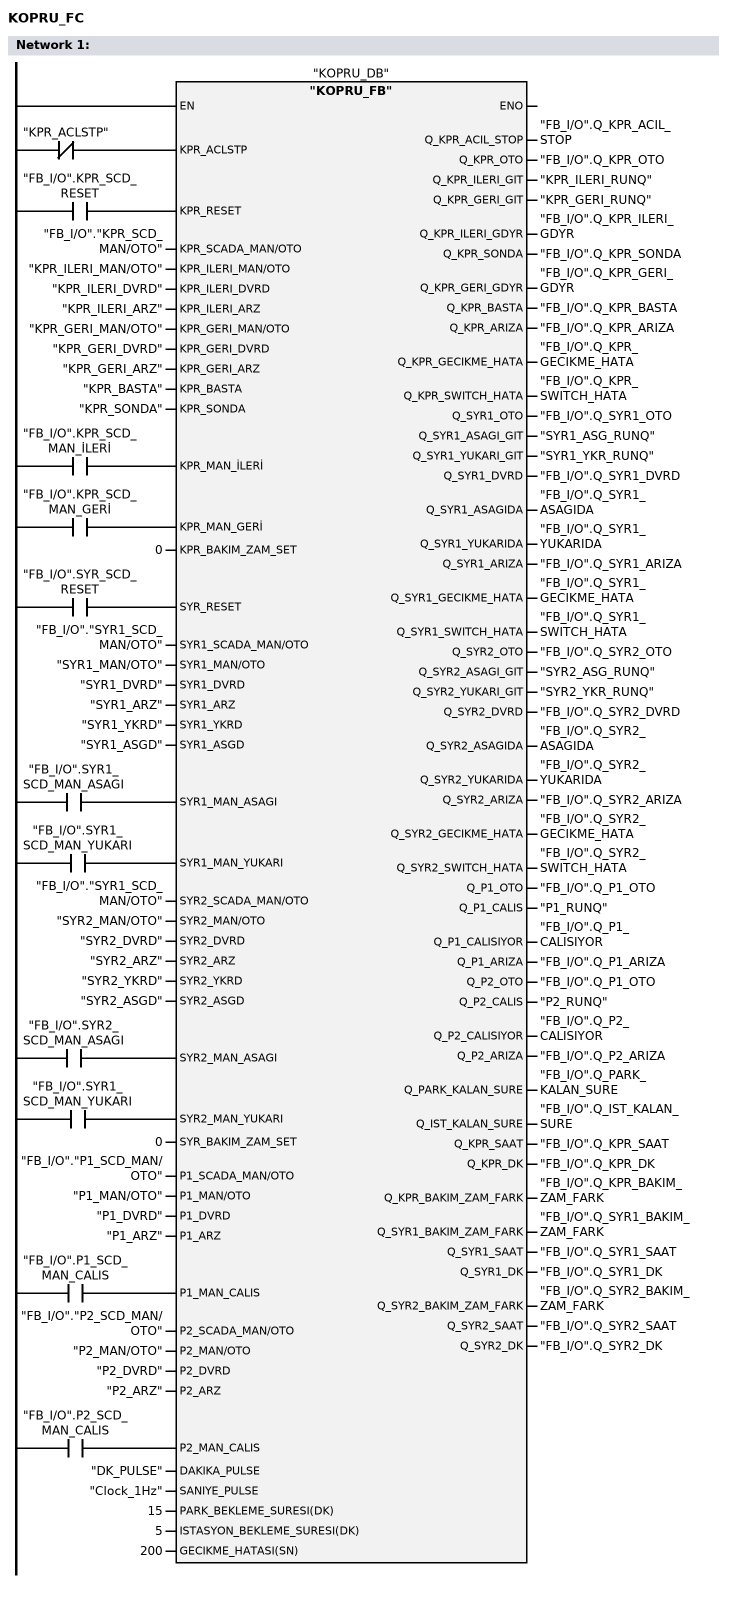
   RUNG wire#powerrail
      "KOPRU_DB"(KPR_ACLSTP := wire#w1, KPR_RESET := wire#w2, KPR_MAN_İLERİ := wire#w3, KPR_MAN_GERİ := wire#w4, SYR_RESET := wire#w5, SYR1_MAN_ASAGI := wire#w6, SYR1_MAN_YUKARI := wire#w7, SYR2_MAN_ASAGI := wire#w8, SYR2_MAN_YUKARI := wire#w9, P1_MAN_CALIS := wire#w10, P2_MAN_CALIS := wire#w11, "KPR_SCADA_MAN/OTO" := "FB_I/O"."KPR_SCD_MAN/OTO", "KPR_ILERI_MAN/OTO" := "KPR_ILERI_MAN/OTO", KPR_ILERI_DVRD := "KPR_ILERI_DVRD", KPR_ILERI_ARZ := "KPR_ILERI_ARZ", "KPR_GERI_MAN/OTO" := "KPR_GERI_MAN/OTO", KPR_GERI_DVRD := "KPR_GERI_DVRD", KPR_GERI_ARZ := "KPR_GERI_ARZ", KPR_BASTA := "KPR_BASTA", KPR_SONDA := "KPR_SONDA", KPR_BAKIM_ZAM_SET := 0, "SYR1_SCADA_MAN/OTO" := "FB_I/O"."SYR1_SCD_MAN/OTO", "SYR1_MAN/OTO" := "SYR1_MAN/OTO", SYR1_DVRD := "SYR1_DVRD", SYR1_ARZ := "SYR1_ARZ", SYR1_YKRD := "SYR1_YKRD", SYR1_ASGD := "SYR1_ASGD", "SYR2_SCADA_MAN/OTO" := "FB_I/O"."SYR1_SCD_MAN/OTO", "SYR2_MAN/OTO" := "SYR2_MAN/OTO", SYR2_DVRD := "SYR2_DVRD", SYR2_ARZ := "SYR2_ARZ", SYR2_YKRD := "SYR2_YKRD", SYR2_ASGD := "SYR2_ASGD", SYR_BAKIM_ZAM_SET := 0, "P1_SCADA_MAN/OTO" := "FB_I/O"."P1_SCD_MAN/OTO", "P1_MAN/OTO" := "P1_MAN/OTO", P1_DVRD := "P1_DVRD", P1_ARZ := "P1_ARZ", "P2_SCADA_MAN/OTO" := "FB_I/O"."P2_SCD_MAN/OTO", "P2_MAN/OTO" := "P2_MAN/OTO", P2_DVRD := "P2_DVRD", P2_ARZ := "P2_ARZ", DAKIKA_PULSE := "DK_PULSE", SANIYE_PULSE := "Clock_1Hz", "PARK_BEKLEME_SURESI(DK)" := 15, "ISTASYON_BEKLEME_SURESI(DK)" := 5, "GECIKME_HATASI(SN)" := 200, Q_KPR_ACIL_STOP => "FB_I/O".Q_KPR_ACIL_STOP, Q_KPR_OTO => "FB_I/O".Q_KPR_OTO, Q_KPR_ILERI_GIT => "KPR_ILERI_RUNQ", Q_KPR_GERI_GIT => "KPR_GERI_RUNQ", Q_KPR_ILERI_GDYR => "FB_I/O".Q_KPR_ILERI_GDYR, Q_KPR_SONDA => "FB_I/O".Q_KPR_SONDA, Q_KPR_GERI_GDYR => "FB_I/O".Q_KPR_GERI_GDYR, Q_KPR_BASTA => "FB_I/O".Q_KPR_BASTA, Q_KPR_ARIZA => "FB_I/O".Q_KPR_ARIZA, Q_KPR_GECIKME_HATA => "FB_I/O".Q_KPR_GECIKME_HATA, Q_KPR_SWITCH_HATA => "FB_I/O".Q_KPR_SWITCH_HATA, Q_SYR1_OTO => "FB_I/O".Q_SYR1_OTO, Q_SYR1_ASAGI_GIT => "SYR1_ASG_RUNQ", Q_SYR1_YUKARI_GIT => "SYR1_YKR_RUNQ", Q_SYR1_DVRD => "FB_I/O".Q_SYR1_DVRD, Q_SYR1_ASAGIDA => "FB_I/O".Q_SYR1_ASAGIDA, Q_SYR1_YUKARIDA => "FB_I/O".Q_SYR1_YUKARIDA, Q_SYR1_ARIZA => "FB_I/O".Q_SYR1_ARIZA, Q_SYR1_GECIKME_HATA => "FB_I/O".Q_SYR1_GECIKME_HATA, Q_SYR1_SWITCH_HATA => "FB_I/O".Q_SYR1_SWITCH_HATA, Q_SYR2_OTO => "FB_I/O".Q_SYR2_OTO, Q_SYR2_ASAGI_GIT => "SYR2_ASG_RUNQ", Q_SYR2_YUKARI_GIT => "SYR2_YKR_RUNQ", Q_SYR2_DVRD => "FB_I/O".Q_SYR2_DVRD, Q_SYR2_ASAGIDA => "FB_I/O".Q_SYR2_ASAGIDA, Q_SYR2_YUKARIDA => "FB_I/O".Q_SYR2_YUKARIDA, Q_SYR2_ARIZA => "FB_I/O".Q_SYR2_ARIZA, Q_SYR2_GECIKME_HATA => "FB_I/O".Q_SYR2_GECIKME_HATA, Q_SYR2_SWITCH_HATA => "FB_I/O".Q_SYR2_SWITCH_HATA, Q_P1_OTO => "FB_I/O".Q_P1_OTO, Q_P1_CALIS => "P1_RUNQ", Q_P1_CALISIYOR => "FB_I/O".Q_P1_CALISIYOR, Q_P1_ARIZA => "FB_I/O".Q_P1_ARIZA, Q_P2_OTO => "FB_I/O".Q_P1_OTO, Q_P2_CALIS => "P2_RUNQ", Q_P2_CALISIYOR => "FB_I/O".Q_P2_CALISIYOR, Q_P2_ARIZA => "FB_I/O".Q_P2_ARIZA, Q_PARK_KALAN_SURE => "FB_I/O".Q_PARK_KALAN_SURE, Q_IST_KALAN_SURE => "FB_I/O".Q_IST_KALAN_SURE, Q_KPR_SAAT => "FB_I/O".Q_KPR_SAAT, Q_KPR_DK => "FB_I/O".Q_KPR_DK, Q_KPR_BAKIM_ZAM_FARK => "FB_I/O".Q_KPR_BAKIM_ZAM_FARK, Q_SYR1_BAKIM_ZAM_FARK => "FB_I/O".Q_SYR1_BAKIM_ZAM_FARK, Q_SYR1_SAAT => "FB_I/O".Q_SYR1_SAAT, Q_SYR1_DK => "FB_I/O".Q_SYR1_DK, Q_SYR2_BAKIM_ZAM_FARK => "FB_I/O".Q_SYR2_BAKIM_ZAM_FARK, Q_SYR2_SAAT => "FB_I/O".Q_SYR2_SAAT, Q_SYR2_DK => "FB_I/O".Q_SYR2_DK)
   END_RUNG
   RUNG wire#powerrail
      I_Contact( "KPR_ACLSTP" )
   END_RUNG wire#w1
   RUNG wire#powerrail
      Contact( "FB_I/O".KPR_SCD_RESET )
   END_RUNG wire#w2
   RUNG wire#powerrail
      Contact( "FB_I/O".KPR_SCD_MAN_İLERİ )
   END_RUNG wire#w3
   RUNG wire#powerrail
      Contact( "FB_I/O".KPR_SCD_MAN_GERİ )
   END_RUNG wire#w4
   RUNG wire#powerrail
      Contact( "FB_I/O".SYR_SCD_RESET )
   END_RUNG wire#w5
   RUNG wire#powerrail
      Contact( "FB_I/O".SYR1_SCD_MAN_ASAGI )
   END_RUNG wire#w6
   RUNG wire#powerrail
      Contact( "FB_I/O".SYR1_SCD_MAN_YUKARI )
   END_RUNG wire#w7
   RUNG wire#powerrail
      Contact( "FB_I/O".SYR2_SCD_MAN_ASAGI )
   END_RUNG wire#w8
   RUNG wire#powerrail
      Contact( "FB_I/O".SYR1_SCD_MAN_YUKARI )
   END_RUNG wire#w9
   RUNG wire#powerrail
      Contact( "FB_I/O".P1_SCD_MAN_CALIS )
   END_RUNG wire#w10
   RUNG wire#powerrail
      Contact( "FB_I/O".P2_SCD_MAN_CALIS )
   END_RUNG wire#w11
   // the same network as SCL:
   "KOPRU_DB"(KPR_ACLSTP := NOT "KPR_ACLSTP",   // "KOPRU_FB"
              KPR_RESET := "FB_I/O".KPR_SCD_RESET,
              "KPR_SCADA_MAN/OTO" := "FB_I/O"."KPR_SCD_MAN/OTO",
              "KPR_ILERI_MAN/OTO" := "KPR_ILERI_MAN/OTO",
              KPR_ILERI_DVRD := "KPR_ILERI_DVRD",
              KPR_ILERI_ARZ := "KPR_ILERI_ARZ",
              "KPR_GERI_MAN/OTO" := "KPR_GERI_MAN/OTO",
              KPR_GERI_DVRD := "KPR_GERI_DVRD",
              KPR_GERI_ARZ := "KPR_GERI_ARZ",
              KPR_BASTA := "KPR_BASTA",
              KPR_SONDA := "KPR_SONDA",
              KPR_MAN_İLERİ := "FB_I/O".KPR_SCD_MAN_İLERİ,
              KPR_MAN_GERİ := "FB_I/O".KPR_SCD_MAN_GERİ,
              KPR_BAKIM_ZAM_SET := 0,
              SYR_RESET := "FB_I/O".SYR_SCD_RESET,
              "SYR1_SCADA_MAN/OTO" := "FB_I/O"."SYR1_SCD_MAN/OTO",
              "SYR1_MAN/OTO" := "SYR1_MAN/OTO",
              SYR1_DVRD := "SYR1_DVRD",
              SYR1_ARZ := "SYR1_ARZ",
              SYR1_YKRD := "SYR1_YKRD",
              SYR1_ASGD := "SYR1_ASGD",
              SYR1_MAN_ASAGI := "FB_I/O".SYR1_SCD_MAN_ASAGI,
              SYR1_MAN_YUKARI := "FB_I/O".SYR1_SCD_MAN_YUKARI,
              "SYR2_SCADA_MAN/OTO" := "FB_I/O"."SYR1_SCD_MAN/OTO",
              "SYR2_MAN/OTO" := "SYR2_MAN/OTO",
              SYR2_DVRD := "SYR2_DVRD",
              SYR2_ARZ := "SYR2_ARZ",
              SYR2_YKRD := "SYR2_YKRD",
              SYR2_ASGD := "SYR2_ASGD",
              SYR2_MAN_ASAGI := "FB_I/O".SYR2_SCD_MAN_ASAGI,
              SYR2_MAN_YUKARI := "FB_I/O".SYR1_SCD_MAN_YUKARI,
              SYR_BAKIM_ZAM_SET := 0,
              "P1_SCADA_MAN/OTO" := "FB_I/O"."P1_SCD_MAN/OTO",
              "P1_MAN/OTO" := "P1_MAN/OTO",
              P1_DVRD := "P1_DVRD",
              P1_ARZ := "P1_ARZ",
              P1_MAN_CALIS := "FB_I/O".P1_SCD_MAN_CALIS,
              "P2_SCADA_MAN/OTO" := "FB_I/O"."P2_SCD_MAN/OTO",
              "P2_MAN/OTO" := "P2_MAN/OTO",
              P2_DVRD := "P2_DVRD",
              P2_ARZ := "P2_ARZ",
              P2_MAN_CALIS := "FB_I/O".P2_SCD_MAN_CALIS,
              DAKIKA_PULSE := "DK_PULSE",
              SANIYE_PULSE := "Clock_1Hz",
              "PARK_BEKLEME_SURESI(DK)" := 15,
              "ISTASYON_BEKLEME_SURESI(DK)" := 5,
              "GECIKME_HATASI(SN)" := 200,
              Q_KPR_ACIL_STOP => "FB_I/O".Q_KPR_ACIL_STOP,
              Q_KPR_OTO => "FB_I/O".Q_KPR_OTO,
              Q_KPR_ILERI_GIT => "KPR_ILERI_RUNQ",
              Q_KPR_GERI_GIT => "KPR_GERI_RUNQ",
              Q_KPR_ILERI_GDYR => "FB_I/O".Q_KPR_ILERI_GDYR,
              Q_KPR_SONDA => "FB_I/O".Q_KPR_SONDA,
              Q_KPR_GERI_GDYR => "FB_I/O".Q_KPR_GERI_GDYR,
              Q_KPR_BASTA => "FB_I/O".Q_KPR_BASTA,
              Q_KPR_ARIZA => "FB_I/O".Q_KPR_ARIZA,
              Q_KPR_GECIKME_HATA => "FB_I/O".Q_KPR_GECIKME_HATA,
              Q_KPR_SWITCH_HATA => "FB_I/O".Q_KPR_SWITCH_HATA,
              Q_SYR1_OTO => "FB_I/O".Q_SYR1_OTO,
              Q_SYR1_ASAGI_GIT => "SYR1_ASG_RUNQ",
              Q_SYR1_YUKARI_GIT => "SYR1_YKR_RUNQ",
              Q_SYR1_DVRD => "FB_I/O".Q_SYR1_DVRD,
              Q_SYR1_ASAGIDA => "FB_I/O".Q_SYR1_ASAGIDA,
              Q_SYR1_YUKARIDA => "FB_I/O".Q_SYR1_YUKARIDA,
              Q_SYR1_ARIZA => "FB_I/O".Q_SYR1_ARIZA,
              Q_SYR1_GECIKME_HATA => "FB_I/O".Q_SYR1_GECIKME_HATA,
              Q_SYR1_SWITCH_HATA => "FB_I/O".Q_SYR1_SWITCH_HATA,
              Q_SYR2_OTO => "FB_I/O".Q_SYR2_OTO,
              Q_SYR2_ASAGI_GIT => "SYR2_ASG_RUNQ",
              Q_SYR2_YUKARI_GIT => "SYR2_YKR_RUNQ",
              Q_SYR2_DVRD => "FB_I/O".Q_SYR2_DVRD,
              Q_SYR2_ASAGIDA => "FB_I/O".Q_SYR2_ASAGIDA,
              Q_SYR2_YUKARIDA => "FB_I/O".Q_SYR2_YUKARIDA,
              Q_SYR2_ARIZA => "FB_I/O".Q_SYR2_ARIZA,
              Q_SYR2_GECIKME_HATA => "FB_I/O".Q_SYR2_GECIKME_HATA,
              Q_SYR2_SWITCH_HATA => "FB_I/O".Q_SYR2_SWITCH_HATA,
              Q_P1_OTO => "FB_I/O".Q_P1_OTO,
              Q_P1_CALIS => "P1_RUNQ",
              Q_P1_CALISIYOR => "FB_I/O".Q_P1_CALISIYOR,
              Q_P1_ARIZA => "FB_I/O".Q_P1_ARIZA,
              Q_P2_OTO => "FB_I/O".Q_P1_OTO,
              Q_P2_CALIS => "P2_RUNQ",
              Q_P2_CALISIYOR => "FB_I/O".Q_P2_CALISIYOR,
              Q_P2_ARIZA => "FB_I/O".Q_P2_ARIZA,
              Q_PARK_KALAN_SURE => "FB_I/O".Q_PARK_KALAN_SURE,
              Q_IST_KALAN_SURE => "FB_I/O".Q_IST_KALAN_SURE,
              Q_KPR_SAAT => "FB_I/O".Q_KPR_SAAT,
              Q_KPR_DK => "FB_I/O".Q_KPR_DK,
              Q_KPR_BAKIM_ZAM_FARK => "FB_I/O".Q_KPR_BAKIM_ZAM_FARK,
              Q_SYR1_BAKIM_ZAM_FARK => "FB_I/O".Q_SYR1_BAKIM_ZAM_FARK,
              Q_SYR1_SAAT => "FB_I/O".Q_SYR1_SAAT,
              Q_SYR1_DK => "FB_I/O".Q_SYR1_DK,
              Q_SYR2_BAKIM_ZAM_FARK => "FB_I/O".Q_SYR2_BAKIM_ZAM_FARK,
              Q_SYR2_SAAT => "FB_I/O".Q_SYR2_SAAT,
              Q_SYR2_DK => "FB_I/O".Q_SYR2_DK);
END_REGION
END_FUNCTION